  PROC DrawPart12()
    MoveL Offs(pOrigin,114.48,92.02,0.00),v60,z0,tPen\WObj:=wPaper;
    MoveL Offs(pOrigin,115.12,91.91,0.00),v40,z0,tPen\WObj:=wPaper;
    MoveL Offs(pOrigin,117.03,89.57,0.00),v40,z0,tPen\WObj:=wPaper;
    MoveL Offs(pOrigin,121.07,85.96,0.00),v40,z0,tPen\WObj:=wPaper;
    MoveL Offs(pOrigin,120.75,85.22,0.00),v40,z0,tPen\WObj:=wPaper;
    MoveL Offs(pOrigin,121.28,84.47,0.00),v40,fine,tPen\WObj:=wPaper;
    MoveL Offs(pOrigin,121.28,84.47,6.00),v60,z5,tPen\WObj:=wPaper;
    MoveL Offs(pOrigin,128.51,83.73,6.00),vTravel,z5,tPen\WObj:=wPaper;
    MoveL Offs(pOrigin,128.51,83.73,0.00),v60,z0,tPen\WObj:=wPaper;
    MoveL Offs(pOrigin,131.80,86.49,0.00),v40,z0,tPen\WObj:=wPaper;
    MoveL Offs(pOrigin,134.03,89.36,0.00),v40,fine,tPen\WObj:=wPaper;
    MoveL Offs(pOrigin,134.03,89.36,6.00),v60,z5,tPen\WObj:=wPaper;
    MoveL Offs(pOrigin,132.23,86.92,6.00),vTravel,z5,tPen\WObj:=wPaper;
    MoveL Offs(pOrigin,132.23,86.92,0.00),v60,z0,tPen\WObj:=wPaper;
    MoveL Offs(pOrigin,132.54,87.24,0.00),v40,z0,tPen\WObj:=wPaper;
    MoveL Offs(pOrigin,132.23,86.92,0.00),v40,fine,tPen\WObj:=wPaper;
    MoveL Offs(pOrigin,132.23,86.92,6.00),v60,z5,tPen\WObj:=wPaper;
    MoveL Offs(pOrigin,137.11,89.89,6.00),vTravel,z5,tPen\WObj:=wPaper;
    MoveL Offs(pOrigin,137.11,89.89,0.00),v60,z0,tPen\WObj:=wPaper;
    MoveL Offs(pOrigin,137.75,90.74,0.00),v40,fine,tPen\WObj:=wPaper;
    MoveL Offs(pOrigin,137.75,90.74,6.00),v60,z5,tPen\WObj:=wPaper;
    MoveL Offs(pOrigin,134.77,96.91,6.00),vTravel,z5,tPen\WObj:=wPaper;
    MoveL Offs(pOrigin,134.77,96.91,0.00),v60,z0,tPen\WObj:=wPaper;
    MoveL Offs(pOrigin,130.74,95.21,0.00),v40,fine,tPen\WObj:=wPaper;
    MoveL Offs(pOrigin,130.74,95.21,6.00),v60,z5,tPen\WObj:=wPaper;
    MoveL Offs(pOrigin,131.06,119.64,6.00),vTravel,z5,tPen\WObj:=wPaper;
    MoveL Offs(pOrigin,131.06,119.64,0.00),v60,z0,tPen\WObj:=wPaper;
    MoveL Offs(pOrigin,131.48,121.34,0.00),v40,z0,tPen\WObj:=wPaper;
    MoveL Offs(pOrigin,131.27,121.03,0.00),v40,z0,tPen\WObj:=wPaper;
    MoveL Offs(pOrigin,131.69,121.34,0.00),v40,z0,tPen\WObj:=wPaper;
    MoveL Offs(pOrigin,132.65,121.34,0.00),v40,z0,tPen\WObj:=wPaper;
    MoveL Offs(pOrigin,132.65,121.34,0.00),v40,z0,tPen\WObj:=wPaper;
    MoveL Offs(pOrigin,133.07,122.62,0.00),v40,z0,tPen\WObj:=wPaper;
    MoveL Offs(pOrigin,132.44,122.94,0.00),v40,fine,tPen\WObj:=wPaper;
    MoveL Offs(pOrigin,132.44,122.94,6.00),v60,z5,tPen\WObj:=wPaper;
    MoveL Offs(pOrigin,130.74,123.04,6.00),vTravel,z5,tPen\WObj:=wPaper;
    MoveL Offs(pOrigin,130.74,123.04,0.00),v60,z0,tPen\WObj:=wPaper;
    MoveL Offs(pOrigin,130.84,121.77,0.00),v40,z0,tPen\WObj:=wPaper;
    MoveL Offs(pOrigin,130.42,121.56,0.00),v40,z0,tPen\WObj:=wPaper;
    MoveL Offs(pOrigin,130.42,121.56,0.00),v40,z0,tPen\WObj:=wPaper;
    MoveL Offs(pOrigin,129.04,121.66,0.00),v40,fine,tPen\WObj:=wPaper;
    MoveL Offs(pOrigin,129.04,121.66,6.00),v60,z5,tPen\WObj:=wPaper;
    MoveL Offs(pOrigin,127.66,121.66,6.00),vTravel,z5,tPen\WObj:=wPaper;
    MoveL Offs(pOrigin,127.66,121.66,0.00),v60,z0,tPen\WObj:=wPaper;
    MoveL Offs(pOrigin,127.62,120.28,0.00),v40,z0,tPen\WObj:=wPaper;
    MoveL Offs(pOrigin,126.91,120.39,0.00),v40,z0,tPen\WObj:=wPaper;
    MoveL Offs(pOrigin,126.91,120.39,0.00),v40,z0,tPen\WObj:=wPaper;
    MoveL Offs(pOrigin,126.91,121.77,0.00),v40,z0,tPen\WObj:=wPaper;
    MoveL Offs(pOrigin,126.91,121.77,0.00),v40,z0,tPen\WObj:=wPaper;
    MoveL Offs(pOrigin,125.64,121.66,0.00),v40,z0,tPen\WObj:=wPaper;
    MoveL Offs(pOrigin,125.64,121.66,0.00),v40,z0,tPen\WObj:=wPaper;
    MoveL Offs(pOrigin,125.60,121.03,0.00),v40,z0,tPen\WObj:=wPaper;
    MoveL Offs(pOrigin,124.68,120.00,0.00),v40,z0,tPen\WObj:=wPaper;
    MoveL Offs(pOrigin,124.29,120.07,0.00),v40,z0,tPen\WObj:=wPaper;
    MoveL Offs(pOrigin,124.04,121.13,0.00),v40,z0,tPen\WObj:=wPaper;
    MoveL Offs(pOrigin,124.26,121.24,0.00),v40,z0,tPen\WObj:=wPaper;
    MoveL Offs(pOrigin,125.64,121.66,0.00),v40,z0,tPen\WObj:=wPaper;
    MoveL Offs(pOrigin,125.64,120.92,0.00),v40,z0,tPen\WObj:=wPaper;
    MoveL Offs(pOrigin,126.28,120.32,0.00),v40,z0,tPen\WObj:=wPaper;
    MoveL Offs(pOrigin,126.91,120.39,0.00),v40,fine,tPen\WObj:=wPaper;
    MoveL Offs(pOrigin,126.91,120.39,6.00),v60,z5,tPen\WObj:=wPaper;
    MoveL Offs(pOrigin,125.64,120.92,6.00),vTravel,z5,tPen\WObj:=wPaper;
    MoveL Offs(pOrigin,125.64,120.92,0.00),v60,z0,tPen\WObj:=wPaper;
    MoveL Offs(pOrigin,124.89,120.18,0.00),v40,fine,tPen\WObj:=wPaper;
    MoveL Offs(pOrigin,124.89,120.18,6.00),v60,z5,tPen\WObj:=wPaper;
    MoveL Offs(pOrigin,124.47,121.56,6.00),vTravel,z5,tPen\WObj:=wPaper;
    MoveL Offs(pOrigin,124.47,121.56,0.00),v60,z0,tPen\WObj:=wPaper;
    MoveL Offs(pOrigin,123.51,122.62,0.00),v40,z0,tPen\WObj:=wPaper;
    MoveL Offs(pOrigin,123.41,122.62,0.00),v40,z0,tPen\WObj:=wPaper;
    MoveL Offs(pOrigin,121.49,122.19,0.00),v40,z0,tPen\WObj:=wPaper;
    MoveL Offs(pOrigin,120.22,121.17,0.00),v40,z0,tPen\WObj:=wPaper;
    MoveL Offs(pOrigin,119.69,121.13,0.00),v40,z0,tPen\WObj:=wPaper;
    MoveL Offs(pOrigin,119.69,121.13,0.00),v40,z0,tPen\WObj:=wPaper;
    MoveL Offs(pOrigin,120.11,121.88,0.00),v40,z0,tPen\WObj:=wPaper;
    MoveL Offs(pOrigin,119.90,122.90,0.00),v40,z0,tPen\WObj:=wPaper;
    MoveL Offs(pOrigin,118.41,123.47,0.00),v40,z0,tPen\WObj:=wPaper;
    MoveL Offs(pOrigin,117.35,123.15,0.00),v40,z0,tPen\WObj:=wPaper;
    MoveL Offs(pOrigin,116.22,123.93,0.00),v40,z0,tPen\WObj:=wPaper;
    MoveL Offs(pOrigin,115.97,125.17,0.00),v40,z0,tPen\WObj:=wPaper;
    MoveL Offs(pOrigin,116.61,126.76,0.00),v40,fine,tPen\WObj:=wPaper;
    MoveL Offs(pOrigin,116.61,126.76,6.00),v60,z5,tPen\WObj:=wPaper;
    MoveL Offs(pOrigin,115.65,125.70,6.00),vTravel,z5,tPen\WObj:=wPaper;
    MoveL Offs(pOrigin,115.65,125.70,0.00),v60,z0,tPen\WObj:=wPaper;
    MoveL Offs(pOrigin,111.61,119.54,0.00),v40,fine,tPen\WObj:=wPaper;
    MoveL Offs(pOrigin,111.61,119.54,6.00),v60,z5,tPen\WObj:=wPaper;
    MoveL Offs(pOrigin,114.27,118.79,6.00),vTravel,z5,tPen\WObj:=wPaper;
    MoveL Offs(pOrigin,114.27,118.79,0.00),v60,z0,tPen\WObj:=wPaper;
    MoveL Offs(pOrigin,114.69,119.25,0.00),v40,z0,tPen\WObj:=wPaper;
    MoveL Offs(pOrigin,115.97,119.57,0.00),v40,z0,tPen\WObj:=wPaper;
    MoveL Offs(pOrigin,116.71,120.28,0.00),v40,z0,tPen\WObj:=wPaper;
    MoveL Offs(pOrigin,116.71,120.28,0.00),v40,z0,tPen\WObj:=wPaper;
    MoveL Offs(pOrigin,117.35,120.28,0.00),v40,z0,tPen\WObj:=wPaper;
    MoveL Offs(pOrigin,117.67,120.71,0.00),v40,z0,tPen\WObj:=wPaper;
    MoveL Offs(pOrigin,117.67,120.71,0.00),v40,z0,tPen\WObj:=wPaper;
    MoveL Offs(pOrigin,118.94,120.81,0.00),v40,z0,tPen\WObj:=wPaper;
    MoveL Offs(pOrigin,119.58,120.32,0.00),v40,z0,tPen\WObj:=wPaper;
    MoveL Offs(pOrigin,119.51,119.54,0.00),v40,z0,tPen\WObj:=wPaper;
    MoveL Offs(pOrigin,119.90,119.50,0.00),v40,z0,tPen\WObj:=wPaper;
    MoveL Offs(pOrigin,119.97,119.96,0.00),v40,z0,tPen\WObj:=wPaper;
    MoveL Offs(pOrigin,119.58,120.32,0.00),v40,z0,tPen\WObj:=wPaper;
    MoveL Offs(pOrigin,120.01,119.54,0.00),v40,z0,tPen\WObj:=wPaper;
    MoveL Offs(pOrigin,120.79,119.75,0.00),v40,z0,tPen\WObj:=wPaper;
    MoveL Offs(pOrigin,120.75,120.81,0.00),v40,fine,tPen\WObj:=wPaper;
    MoveL Offs(pOrigin,120.75,120.81,6.00),v60,z5,tPen\WObj:=wPaper;
    MoveL Offs(pOrigin,118.31,119.11,6.00),vTravel,z5,tPen\WObj:=wPaper;
    MoveL Offs(pOrigin,118.31,119.11,0.00),v60,z0,tPen\WObj:=wPaper;
    MoveL Offs(pOrigin,117.46,120.28,0.00),v40,fine,tPen\WObj:=wPaper;
    MoveL Offs(pOrigin,117.46,120.28,6.00),v60,z5,tPen\WObj:=wPaper;
    MoveL Offs(pOrigin,117.03,118.26,6.00),vTravel,z5,tPen\WObj:=wPaper;
    MoveL Offs(pOrigin,117.03,118.26,0.00),v60,z0,tPen\WObj:=wPaper;
    MoveL Offs(pOrigin,116.29,117.73,0.00),v40,z0,tPen\WObj:=wPaper;
    MoveL Offs(pOrigin,115.44,117.73,0.00),v40,z0,tPen\WObj:=wPaper;
    MoveL Offs(pOrigin,114.27,118.79,0.00),v40,z0,tPen\WObj:=wPaper;
    MoveL Offs(pOrigin,114.27,118.79,0.00),v40,z0,tPen\WObj:=wPaper;
    MoveL Offs(pOrigin,113.21,117.94,0.00),v40,z0,tPen\WObj:=wPaper;
    MoveL Offs(pOrigin,113.74,116.03,0.00),v40,fine,tPen\WObj:=wPaper;
    MoveL Offs(pOrigin,113.74,116.03,6.00),v60,z5,tPen\WObj:=wPaper;
    MoveL Offs(pOrigin,116.61,117.84,6.00),vTravel,z5,tPen\WObj:=wPaper;
    MoveL Offs(pOrigin,116.61,117.84,0.00),v60,z0,tPen\WObj:=wPaper;
    MoveL Offs(pOrigin,130.21,119.32,0.00),v40,z0,tPen\WObj:=wPaper;
  ENDPROC

  PROC DrawPart13()
    MoveL Offs(pOrigin,131.80,119.68,0.00),v40,z0,tPen\WObj:=wPaper;
    MoveL Offs(pOrigin,132.76,120.71,0.00),v40,z0,tPen\WObj:=wPaper;
    MoveL Offs(pOrigin,132.76,120.71,0.00),v40,z0,tPen\WObj:=wPaper;
    MoveL Offs(pOrigin,131.80,119.75,0.00),v40,fine,tPen\WObj:=wPaper;
    MoveL Offs(pOrigin,131.80,119.75,6.00),v60,z5,tPen\WObj:=wPaper;
    MoveL Offs(pOrigin,134.56,122.41,6.00),vTravel,z5,tPen\WObj:=wPaper;
    MoveL Offs(pOrigin,134.56,122.41,0.00),v60,z0,tPen\WObj:=wPaper;
    MoveL Offs(pOrigin,128.61,127.40,0.00),v40,z0,tPen\WObj:=wPaper;
    MoveL Offs(pOrigin,127.55,127.72,0.00),v40,z0,tPen\WObj:=wPaper;
    MoveL Offs(pOrigin,128.19,126.12,0.00),v40,z0,tPen\WObj:=wPaper;
    MoveL Offs(pOrigin,127.90,125.06,0.00),v40,z0,tPen\WObj:=wPaper;
    MoveL Offs(pOrigin,127.23,124.39,0.00),v40,z0,tPen\WObj:=wPaper;
    MoveL Offs(pOrigin,126.38,124.32,0.00),v40,z0,tPen\WObj:=wPaper;
    MoveL Offs(pOrigin,126.38,124.32,0.00),v40,z0,tPen\WObj:=wPaper;
    MoveL Offs(pOrigin,126.06,124.64,0.00),v40,z0,tPen\WObj:=wPaper;
    MoveL Offs(pOrigin,125.00,124.25,0.00),v40,z0,tPen\WObj:=wPaper;
    MoveL Offs(pOrigin,123.51,122.72,0.00),v40,z0,tPen\WObj:=wPaper;
    MoveL Offs(pOrigin,123.94,123.47,0.00),v40,z0,tPen\WObj:=wPaper;
    MoveL Offs(pOrigin,124.26,123.79,0.00),v40,z0,tPen\WObj:=wPaper;
    MoveL Offs(pOrigin,123.94,123.47,0.00),v40,fine,tPen\WObj:=wPaper;
    MoveL Offs(pOrigin,123.94,123.47,6.00),v60,z5,tPen\WObj:=wPaper;
    MoveL Offs(pOrigin,127.66,121.66,6.00),vTravel,z5,tPen\WObj:=wPaper;
    MoveL Offs(pOrigin,127.66,121.66,0.00),v60,z0,tPen\WObj:=wPaper;
    MoveL Offs(pOrigin,129.00,121.77,0.00),v40,z0,tPen\WObj:=wPaper;
    MoveL Offs(pOrigin,129.00,122.51,0.00),v40,z0,tPen\WObj:=wPaper;
    MoveL Offs(pOrigin,128.51,123.26,0.00),v40,fine,tPen\WObj:=wPaper;
    MoveL Offs(pOrigin,128.51,123.26,6.00),v60,z5,tPen\WObj:=wPaper;
    MoveL Offs(pOrigin,129.99,131.76,6.00),vTravel,z5,tPen\WObj:=wPaper;
    MoveL Offs(pOrigin,129.99,131.76,0.00),v60,z0,tPen\WObj:=wPaper;
    MoveL Offs(pOrigin,127.66,132.36,0.00),v40,z0,tPen\WObj:=wPaper;
    MoveL Offs(pOrigin,125.96,133.24,0.00),v40,z0,tPen\WObj:=wPaper;
    MoveL Offs(pOrigin,127.02,133.56,0.00),v40,z0,tPen\WObj:=wPaper;
    MoveL Offs(pOrigin,128.82,133.14,0.00),v40,fine,tPen\WObj:=wPaper;
    MoveL Offs(pOrigin,128.82,133.14,6.00),v60,z5,tPen\WObj:=wPaper;
    MoveL Offs(pOrigin,129.46,135.37,6.00),vTravel,z5,tPen\WObj:=wPaper;
    MoveL Offs(pOrigin,129.46,135.37,0.00),v60,z0,tPen\WObj:=wPaper;
    MoveL Offs(pOrigin,128.75,135.51,0.00),v40,z0,tPen\WObj:=wPaper;
    MoveL Offs(pOrigin,128.72,136.25,0.00),v40,z0,tPen\WObj:=wPaper;
    MoveL Offs(pOrigin,129.78,135.48,0.00),v40,z0,tPen\WObj:=wPaper;
    MoveL Offs(pOrigin,130.52,136.22,0.00),v40,z0,tPen\WObj:=wPaper;
    MoveL Offs(pOrigin,130.10,136.71,0.00),v40,z0,tPen\WObj:=wPaper;
    MoveL Offs(pOrigin,129.14,136.75,0.00),v40,z0,tPen\WObj:=wPaper;
    MoveL Offs(pOrigin,127.87,136.25,0.00),v40,z0,tPen\WObj:=wPaper;
    MoveL Offs(pOrigin,126.81,135.26,0.00),v40,z0,tPen\WObj:=wPaper;
    MoveL Offs(pOrigin,126.81,135.26,0.00),v40,z0,tPen\WObj:=wPaper;
    MoveL Offs(pOrigin,126.91,134.84,0.00),v40,z0,tPen\WObj:=wPaper;
    MoveL Offs(pOrigin,126.38,134.62,0.00),v40,z0,tPen\WObj:=wPaper;
    MoveL Offs(pOrigin,126.91,134.73,0.00),v40,z0,tPen\WObj:=wPaper;
    MoveL Offs(pOrigin,129.04,134.73,0.00),v40,z0,tPen\WObj:=wPaper;
    MoveL Offs(pOrigin,129.57,135.33,0.00),v40,z0,tPen\WObj:=wPaper;
    MoveL Offs(pOrigin,130.38,135.62,0.00),v40,z0,tPen\WObj:=wPaper;
    MoveL Offs(pOrigin,130.52,136.22,0.00),v40,z0,tPen\WObj:=wPaper;
    MoveL Offs(pOrigin,130.52,136.22,0.00),v40,z0,tPen\WObj:=wPaper;
    MoveL Offs(pOrigin,131.48,136.64,0.00),v40,z0,tPen\WObj:=wPaper;
    MoveL Offs(pOrigin,133.18,135.90,0.00),v40,z0,tPen\WObj:=wPaper;
    MoveL Offs(pOrigin,133.93,135.90,0.00),v40,z0,tPen\WObj:=wPaper;
    MoveL Offs(pOrigin,133.93,135.90,0.00),v40,z0,tPen\WObj:=wPaper;
    MoveL Offs(pOrigin,134.46,136.11,0.00),v40,z0,tPen\WObj:=wPaper;
    MoveL Offs(pOrigin,135.20,135.79,0.00),v40,fine,tPen\WObj:=wPaper;
    MoveL Offs(pOrigin,135.20,135.79,6.00),v60,z5,tPen\WObj:=wPaper;
    MoveL Offs(pOrigin,136.37,135.48,6.00),vTravel,z5,tPen\WObj:=wPaper;
    MoveL Offs(pOrigin,136.37,135.48,0.00),v60,z0,tPen\WObj:=wPaper;
    MoveL Offs(pOrigin,134.88,135.37,0.00),v40,z0,tPen\WObj:=wPaper;
    MoveL Offs(pOrigin,133.93,135.90,0.00),v40,z0,tPen\WObj:=wPaper;
    MoveL Offs(pOrigin,133.93,136.11,0.00),v40,z0,tPen\WObj:=wPaper;
    MoveL Offs(pOrigin,133.50,136.68,0.00),v40,z0,tPen\WObj:=wPaper;
    MoveL Offs(pOrigin,132.44,137.18,0.00),v40,z0,tPen\WObj:=wPaper;
    MoveL Offs(pOrigin,128.61,137.49,0.00),v40,z0,tPen\WObj:=wPaper;
    MoveL Offs(pOrigin,127.12,137.14,0.00),v40,z0,tPen\WObj:=wPaper;
    MoveL Offs(pOrigin,125.43,135.48,0.00),v40,z0,tPen\WObj:=wPaper;
    MoveL Offs(pOrigin,124.68,135.16,0.00),v40,z0,tPen\WObj:=wPaper;
    MoveL Offs(pOrigin,124.57,135.37,0.00),v40,z0,tPen\WObj:=wPaper;
    MoveL Offs(pOrigin,125.53,135.79,0.00),v40,fine,tPen\WObj:=wPaper;
    MoveL Offs(pOrigin,125.53,135.79,6.00),v60,z5,tPen\WObj:=wPaper;
    MoveL Offs(pOrigin,123.62,134.41,6.00),vTravel,z5,tPen\WObj:=wPaper;
    MoveL Offs(pOrigin,123.62,134.41,0.00),v60,z0,tPen\WObj:=wPaper;
    MoveL Offs(pOrigin,123.30,135.37,0.00),v40,z0,tPen\WObj:=wPaper;
    MoveL Offs(pOrigin,123.37,136.64,0.00),v40,z0,tPen\WObj:=wPaper;
    MoveL Offs(pOrigin,124.79,137.85,0.00),v40,z0,tPen\WObj:=wPaper;
    MoveL Offs(pOrigin,131.80,139.19,0.00),v40,z0,tPen\WObj:=wPaper;
    MoveL Offs(pOrigin,134.14,139.09,0.00),v40,z0,tPen\WObj:=wPaper;
    MoveL Offs(pOrigin,135.41,138.34,0.00),v40,fine,tPen\WObj:=wPaper;
    MoveL Offs(pOrigin,135.41,138.34,6.00),v60,z5,tPen\WObj:=wPaper;
    MoveL Offs(pOrigin,137.54,138.88,6.00),vTravel,z5,tPen\WObj:=wPaper;
    MoveL Offs(pOrigin,137.54,138.88,0.00),v60,z0,tPen\WObj:=wPaper;
    MoveL Offs(pOrigin,138.18,137.18,0.00),v40,z0,tPen\WObj:=wPaper;
    MoveL Offs(pOrigin,138.18,137.18,0.00),v40,z0,tPen\WObj:=wPaper;
    MoveL Offs(pOrigin,138.18,133.67,0.00),v40,z0,tPen\WObj:=wPaper;
    MoveL Offs(pOrigin,137.43,131.54,0.00),v40,z0,tPen\WObj:=wPaper;
    MoveL Offs(pOrigin,135.52,130.55,0.00),v40,z0,tPen\WObj:=wPaper;
    MoveL Offs(pOrigin,133.18,129.95,0.00),v40,z0,tPen\WObj:=wPaper;
    MoveL Offs(pOrigin,130.10,129.52,0.00),v40,z0,tPen\WObj:=wPaper;
    MoveL Offs(pOrigin,127.44,129.52,0.00),v40,z0,tPen\WObj:=wPaper;
    MoveL Offs(pOrigin,125.96,129.91,0.00),v40,z0,tPen\WObj:=wPaper;
    MoveL Offs(pOrigin,124.04,131.86,0.00),v40,z0,tPen\WObj:=wPaper;
    MoveL Offs(pOrigin,123.26,133.03,0.00),v40,z0,tPen\WObj:=wPaper;
    MoveL Offs(pOrigin,122.63,135.37,0.00),v40,z0,tPen\WObj:=wPaper;
    MoveL Offs(pOrigin,120.96,135.69,0.00),v40,z0,tPen\WObj:=wPaper;
    MoveL Offs(pOrigin,119.05,135.19,0.00),v40,z0,tPen\WObj:=wPaper;
    MoveL Offs(pOrigin,118.62,134.73,0.00),v40,z0,tPen\WObj:=wPaper;
    MoveL Offs(pOrigin,118.84,133.77,0.00),v40,z0,tPen\WObj:=wPaper;
    MoveL Offs(pOrigin,118.84,133.56,0.00),v40,z0,tPen\WObj:=wPaper;
    MoveL Offs(pOrigin,118.73,132.61,0.00),v40,z0,tPen\WObj:=wPaper;
    MoveL Offs(pOrigin,118.73,132.61,0.00),v40,z0,tPen\WObj:=wPaper;
    MoveL Offs(pOrigin,118.31,131.23,0.00),v40,z0,tPen\WObj:=wPaper;
    MoveL Offs(pOrigin,118.31,131.01,0.00),v40,z0,tPen\WObj:=wPaper;
    MoveL Offs(pOrigin,117.46,129.31,0.00),v40,z0,tPen\WObj:=wPaper;
    MoveL Offs(pOrigin,116.07,128.32,0.00),v40,z0,tPen\WObj:=wPaper;
    MoveL Offs(pOrigin,112.78,127.51,0.00),v40,z0,tPen\WObj:=wPaper;
    MoveL Offs(pOrigin,108.53,127.19,0.00),v40,z0,tPen\WObj:=wPaper;
    MoveL Offs(pOrigin,106.72,127.40,0.00),v40,z0,tPen\WObj:=wPaper;
    MoveL Offs(pOrigin,105.45,128.04,0.00),v40,z0,tPen\WObj:=wPaper;
    MoveL Offs(pOrigin,104.46,129.63,0.00),v40,z0,tPen\WObj:=wPaper;
    MoveL Offs(pOrigin,103.54,132.18,0.00),v40,z0,tPen\WObj:=wPaper;
    MoveL Offs(pOrigin,103.54,132.18,0.00),v40,z0,tPen\WObj:=wPaper;
    MoveL Offs(pOrigin,104.07,135.16,0.00),v40,z0,tPen\WObj:=wPaper;
    MoveL Offs(pOrigin,104.07,135.16,0.00),v40,z0,tPen\WObj:=wPaper;
    MoveL Offs(pOrigin,105.34,135.94,0.00),v40,z0,tPen\WObj:=wPaper;
    MoveL Offs(pOrigin,109.17,137.28,0.00),v40,z0,tPen\WObj:=wPaper;
    MoveL Offs(pOrigin,113.74,137.71,0.00),v40,z0,tPen\WObj:=wPaper;
  ENDPROC

  PROC DrawPart14()
    MoveL Offs(pOrigin,115.01,138.24,0.00),v40,z0,tPen\WObj:=wPaper;
    MoveL Offs(pOrigin,114.80,137.49,0.00),v40,z0,tPen\WObj:=wPaper;
    MoveL Offs(pOrigin,117.78,136.75,0.00),v40,z0,tPen\WObj:=wPaper;
    MoveL Offs(pOrigin,117.99,137.07,0.00),v40,z0,tPen\WObj:=wPaper;
    MoveL Offs(pOrigin,117.78,136.64,0.00),v40,z0,tPen\WObj:=wPaper;
    MoveL Offs(pOrigin,118.09,136.32,0.00),v40,z0,tPen\WObj:=wPaper;
    MoveL Offs(pOrigin,118.09,136.32,0.00),v40,z0,tPen\WObj:=wPaper;
    MoveL Offs(pOrigin,118.31,136.75,0.00),v40,z0,tPen\WObj:=wPaper;
    MoveL Offs(pOrigin,117.99,137.28,0.00),v40,z0,tPen\WObj:=wPaper;
    MoveL Offs(pOrigin,118.09,139.62,0.00),v40,fine,tPen\WObj:=wPaper;
    MoveL Offs(pOrigin,118.09,139.62,6.00),v60,z5,tPen\WObj:=wPaper;
    MoveL Offs(pOrigin,118.09,136.32,6.00),vTravel,z5,tPen\WObj:=wPaper;
    MoveL Offs(pOrigin,118.09,136.32,0.00),v60,z0,tPen\WObj:=wPaper;
    MoveL Offs(pOrigin,118.41,135.79,0.00),v40,z0,tPen\WObj:=wPaper;
    MoveL Offs(pOrigin,120.75,136.43,0.00),v40,z0,tPen\WObj:=wPaper;
    MoveL Offs(pOrigin,122.45,136.32,0.00),v40,z0,tPen\WObj:=wPaper;
    MoveL Offs(pOrigin,122.88,137.35,0.00),v40,z0,tPen\WObj:=wPaper;
    MoveL Offs(pOrigin,125.21,139.02,0.00),v40,z0,tPen\WObj:=wPaper;
    MoveL Offs(pOrigin,127.02,139.62,0.00),v40,z0,tPen\WObj:=wPaper;
    MoveL Offs(pOrigin,132.12,140.26,0.00),v40,z0,tPen\WObj:=wPaper;
    MoveL Offs(pOrigin,135.94,139.73,0.00),v40,z0,tPen\WObj:=wPaper;
    MoveL Offs(pOrigin,137.54,138.88,0.00),v40,z0,tPen\WObj:=wPaper;
    MoveL Offs(pOrigin,137.54,138.88,0.00),v40,z0,tPen\WObj:=wPaper;
    MoveL Offs(pOrigin,139.66,139.09,0.00),v40,z0,tPen\WObj:=wPaper;
    MoveL Offs(pOrigin,139.66,139.09,0.00),v40,z0,tPen\WObj:=wPaper;
    MoveL Offs(pOrigin,139.63,138.45,0.00),v40,z0,tPen\WObj:=wPaper;
    MoveL Offs(pOrigin,138.71,138.02,0.00),v40,z0,tPen\WObj:=wPaper;
    MoveL Offs(pOrigin,138.18,137.18,0.00),v40,z0,tPen\WObj:=wPaper;
    MoveL Offs(pOrigin,139.77,137.92,0.00),v40,z0,tPen\WObj:=wPaper;
    MoveL Offs(pOrigin,139.66,138.34,0.00),v40,z0,tPen\WObj:=wPaper;
    MoveL Offs(pOrigin,139.98,137.92,0.00),v40,z0,tPen\WObj:=wPaper;
    MoveL Offs(pOrigin,142.43,137.81,0.00),v40,z0,tPen\WObj:=wPaper;
    MoveL Offs(pOrigin,142.21,138.56,0.00),v40,z0,tPen\WObj:=wPaper;
    MoveL Offs(pOrigin,140.41,138.45,0.00),v40,z0,tPen\WObj:=wPaper;
    MoveL Offs(pOrigin,139.66,139.09,0.00),v40,z0,tPen\WObj:=wPaper;
    MoveL Offs(pOrigin,141.15,139.09,0.00),v40,z0,tPen\WObj:=wPaper;
    MoveL Offs(pOrigin,141.57,139.51,0.00),v40,fine,tPen\WObj:=wPaper;
    MoveL Offs(pOrigin,141.57,139.51,6.00),v60,z5,tPen\WObj:=wPaper;
    MoveL Offs(pOrigin,142.74,140.79,6.00),vTravel,z5,tPen\WObj:=wPaper;
    MoveL Offs(pOrigin,142.74,140.79,0.00),v60,z0,tPen\WObj:=wPaper;
    MoveL Offs(pOrigin,140.94,143.23,0.00),v40,z0,tPen\WObj:=wPaper;
    MoveL Offs(pOrigin,140.94,143.23,0.00),v40,z0,tPen\WObj:=wPaper;
    MoveL Offs(pOrigin,139.66,145.78,0.00),v40,z0,tPen\WObj:=wPaper;
    MoveL Offs(pOrigin,139.45,144.93,0.00),v40,z0,tPen\WObj:=wPaper;
    MoveL Offs(pOrigin,140.41,143.44,0.00),v40,z0,tPen\WObj:=wPaper;
    MoveL Offs(pOrigin,140.94,143.23,0.00),v40,z0,tPen\WObj:=wPaper;
    MoveL Offs(pOrigin,140.73,142.38,0.00),v40,z0,tPen\WObj:=wPaper;
    MoveL Offs(pOrigin,141.15,141.32,0.00),v40,z0,tPen\WObj:=wPaper;
    MoveL Offs(pOrigin,141.15,141.32,0.00),v40,z0,tPen\WObj:=wPaper;
    MoveL Offs(pOrigin,142.43,141.21,0.00),v40,z0,tPen\WObj:=wPaper;
    MoveL Offs(pOrigin,142.74,140.79,0.00),v40,z0,tPen\WObj:=wPaper;
    MoveL Offs(pOrigin,144.44,140.15,0.00),v40,z0,tPen\WObj:=wPaper;
    MoveL Offs(pOrigin,144.44,140.15,0.00),v40,z0,tPen\WObj:=wPaper;
    MoveL Offs(pOrigin,145.40,140.57,0.00),v40,z0,tPen\WObj:=wPaper;
    MoveL Offs(pOrigin,146.36,140.47,0.00),v40,z0,tPen\WObj:=wPaper;
    MoveL Offs(pOrigin,145.82,139.90,0.00),v40,z0,tPen\WObj:=wPaper;
    MoveL Offs(pOrigin,145.08,139.73,0.00),v40,z0,tPen\WObj:=wPaper;
    MoveL Offs(pOrigin,144.44,140.15,0.00),v40,z0,tPen\WObj:=wPaper;
    MoveL Offs(pOrigin,144.66,141.21,0.00),v40,z0,tPen\WObj:=wPaper;
    MoveL Offs(pOrigin,143.27,141.85,0.00),v40,z0,tPen\WObj:=wPaper;
    MoveL Offs(pOrigin,143.17,142.81,0.00),v40,z0,tPen\WObj:=wPaper;
    MoveL Offs(pOrigin,143.17,142.81,0.00),v40,z0,tPen\WObj:=wPaper;
    MoveL Offs(pOrigin,141.68,144.19,0.00),v40,z0,tPen\WObj:=wPaper;
    MoveL Offs(pOrigin,141.47,145.04,0.00),v40,z0,tPen\WObj:=wPaper;
    MoveL Offs(pOrigin,141.47,145.04,0.00),v40,z0,tPen\WObj:=wPaper;
    MoveL Offs(pOrigin,140.65,146.52,0.00),v40,z0,tPen\WObj:=wPaper;
    MoveL Offs(pOrigin,141.26,147.06,0.00),v40,z0,tPen\WObj:=wPaper;
    MoveL Offs(pOrigin,141.26,147.06,0.00),v40,z0,tPen\WObj:=wPaper;
    MoveL Offs(pOrigin,143.27,145.53,0.00),v40,z0,tPen\WObj:=wPaper;
    MoveL Offs(pOrigin,143.59,145.68,0.00),v40,z0,tPen\WObj:=wPaper;
    MoveL Offs(pOrigin,143.49,145.46,0.00),v40,z0,tPen\WObj:=wPaper;
    MoveL Offs(pOrigin,145.93,145.68,0.00),v40,z0,tPen\WObj:=wPaper;
    MoveL Offs(pOrigin,146.46,146.31,0.00),v40,z0,tPen\WObj:=wPaper;
    MoveL Offs(pOrigin,146.46,146.31,0.00),v40,z0,tPen\WObj:=wPaper;
    MoveL Offs(pOrigin,144.23,146.70,0.00),v40,z0,tPen\WObj:=wPaper;
    MoveL Offs(pOrigin,143.31,147.48,0.00),v40,z0,tPen\WObj:=wPaper;
    MoveL Offs(pOrigin,143.70,147.69,0.00),v40,z0,tPen\WObj:=wPaper;
    MoveL Offs(pOrigin,144.76,147.48,0.00),v40,z0,tPen\WObj:=wPaper;
    MoveL Offs(pOrigin,147.10,148.23,0.00),v40,z0,tPen\WObj:=wPaper;
    MoveL Offs(pOrigin,147.10,148.23,0.00),v40,z0,tPen\WObj:=wPaper;
    MoveL Offs(pOrigin,147.21,149.18,0.00),v40,z0,tPen\WObj:=wPaper;
    MoveL Offs(pOrigin,147.21,149.18,0.00),v40,z0,tPen\WObj:=wPaper;
    MoveL Offs(pOrigin,148.16,149.50,0.00),v40,z0,tPen\WObj:=wPaper;
    MoveL Offs(pOrigin,148.16,149.50,0.00),v40,z0,tPen\WObj:=wPaper;
    MoveL Offs(pOrigin,148.45,148.44,0.00),v40,z0,tPen\WObj:=wPaper;
    MoveL Offs(pOrigin,147.10,148.23,0.00),v40,z0,tPen\WObj:=wPaper;
    MoveL Offs(pOrigin,147.21,149.18,0.00),v40,z0,tPen\WObj:=wPaper;
    MoveL Offs(pOrigin,145.08,149.07,0.00),v40,z0,tPen\WObj:=wPaper;
    MoveL Offs(pOrigin,143.81,149.61,0.00),v40,z0,tPen\WObj:=wPaper;
    MoveL Offs(pOrigin,143.81,149.61,0.00),v40,z0,tPen\WObj:=wPaper;
    MoveL Offs(pOrigin,143.91,150.21,0.00),v40,z0,tPen\WObj:=wPaper;
    MoveL Offs(pOrigin,145.51,150.03,0.00),v40,z0,tPen\WObj:=wPaper;
    MoveL Offs(pOrigin,146.25,150.46,0.00),v40,z0,tPen\WObj:=wPaper;
    MoveL Offs(pOrigin,146.25,150.46,0.00),v40,z0,tPen\WObj:=wPaper;
    MoveL Offs(pOrigin,148.27,151.20,0.00),v40,z0,tPen\WObj:=wPaper;
    MoveL Offs(pOrigin,148.27,151.20,0.00),v40,z0,tPen\WObj:=wPaper;
    MoveL Offs(pOrigin,148.06,152.37,0.00),v40,z0,tPen\WObj:=wPaper;
    MoveL Offs(pOrigin,148.06,152.37,0.00),v40,z0,tPen\WObj:=wPaper;
    MoveL Offs(pOrigin,146.89,152.05,0.00),v40,z0,tPen\WObj:=wPaper;
    MoveL Offs(pOrigin,146.68,152.37,0.00),v40,z0,tPen\WObj:=wPaper;
    MoveL Offs(pOrigin,147.21,152.83,0.00),v40,z0,tPen\WObj:=wPaper;
    MoveL Offs(pOrigin,148.06,152.90,0.00),v40,z0,tPen\WObj:=wPaper;
    MoveL Offs(pOrigin,148.06,152.90,0.00),v40,z0,tPen\WObj:=wPaper;
    MoveL Offs(pOrigin,147.84,154.07,0.00),v40,z0,tPen\WObj:=wPaper;
    MoveL Offs(pOrigin,147.84,154.07,0.00),v40,z0,tPen\WObj:=wPaper;
    MoveL Offs(pOrigin,147.56,155.34,0.00),v40,z0,tPen\WObj:=wPaper;
    MoveL Offs(pOrigin,146.78,155.77,0.00),v40,z0,tPen\WObj:=wPaper;
    MoveL Offs(pOrigin,146.53,156.73,0.00),v40,z0,tPen\WObj:=wPaper;
    MoveL Offs(pOrigin,146.07,157.15,0.00),v40,z0,tPen\WObj:=wPaper;
    MoveL Offs(pOrigin,145.93,159.06,0.00),v40,z0,tPen\WObj:=wPaper;
    MoveL Offs(pOrigin,145.40,158.96,0.00),v40,z0,tPen\WObj:=wPaper;
    MoveL Offs(pOrigin,145.44,158.11,0.00),v40,z0,tPen\WObj:=wPaper;
    MoveL Offs(pOrigin,145.93,157.79,0.00),v40,z0,tPen\WObj:=wPaper;
    MoveL Offs(pOrigin,146.04,157.04,0.00),v40,z0,tPen\WObj:=wPaper;
    MoveL Offs(pOrigin,145.51,155.77,0.00),v40,z0,tPen\WObj:=wPaper;
    MoveL Offs(pOrigin,145.51,155.77,0.00),v40,z0,tPen\WObj:=wPaper;
    MoveL Offs(pOrigin,144.94,156.19,0.00),v40,z0,tPen\WObj:=wPaper;
    MoveL Offs(pOrigin,143.56,158.74,0.00),v40,z0,tPen\WObj:=wPaper;
    MoveL Offs(pOrigin,141.89,159.59,0.00),v40,z0,tPen\WObj:=wPaper;
    MoveL Offs(pOrigin,140.09,159.35,0.00),v40,z0,tPen\WObj:=wPaper;
  ENDPROC

  PROC DrawPart15()
    MoveL Offs(pOrigin,137.75,158.00,0.00),v40,z0,tPen\WObj:=wPaper;
    MoveL Offs(pOrigin,135.73,158.00,0.00),v40,z0,tPen\WObj:=wPaper;
    MoveL Offs(pOrigin,135.31,158.32,0.00),v40,z0,tPen\WObj:=wPaper;
    MoveL Offs(pOrigin,135.31,158.32,0.00),v40,z0,tPen\WObj:=wPaper;
    MoveL Offs(pOrigin,132.97,158.21,0.00),v40,z0,tPen\WObj:=wPaper;
    MoveL Offs(pOrigin,130.42,157.36,0.00),v40,fine,tPen\WObj:=wPaper;
    MoveL Offs(pOrigin,130.42,157.36,6.00),v60,z5,tPen\WObj:=wPaper;
    MoveL Offs(pOrigin,129.04,157.68,6.00),vTravel,z5,tPen\WObj:=wPaper;
    MoveL Offs(pOrigin,129.04,157.68,0.00),v60,z0,tPen\WObj:=wPaper;
    MoveL Offs(pOrigin,130.84,158.85,0.00),v40,z0,tPen\WObj:=wPaper;
    MoveL Offs(pOrigin,134.03,159.27,0.00),v40,z0,tPen\WObj:=wPaper;
    MoveL Offs(pOrigin,134.67,160.12,0.00),v40,z0,tPen\WObj:=wPaper;
    MoveL Offs(pOrigin,135.62,160.76,0.00),v40,z0,tPen\WObj:=wPaper;
    MoveL Offs(pOrigin,135.62,160.76,0.00),v40,z0,tPen\WObj:=wPaper;
    MoveL Offs(pOrigin,137.86,161.61,0.00),v40,fine,tPen\WObj:=wPaper;
    MoveL Offs(pOrigin,137.86,161.61,6.00),v60,z5,tPen\WObj:=wPaper;
    MoveL Offs(pOrigin,136.69,162.78,6.00),vTravel,z5,tPen\WObj:=wPaper;
    MoveL Offs(pOrigin,136.69,162.78,0.00),v60,z0,tPen\WObj:=wPaper;
    MoveL Offs(pOrigin,134.46,161.19,0.00),v40,z0,tPen\WObj:=wPaper;
    MoveL Offs(pOrigin,134.46,161.19,0.00),v40,z0,tPen\WObj:=wPaper;
    MoveL Offs(pOrigin,135.52,161.22,0.00),v40,z0,tPen\WObj:=wPaper;
    MoveL Offs(pOrigin,139.56,163.42,0.00),v40,z0,tPen\WObj:=wPaper;
    MoveL Offs(pOrigin,141.86,163.52,0.00),v40,z0,tPen\WObj:=wPaper;
    MoveL Offs(pOrigin,141.75,164.02,0.00),v40,z0,tPen\WObj:=wPaper;
    MoveL Offs(pOrigin,140.30,164.69,0.00),v40,z0,tPen\WObj:=wPaper;
    MoveL Offs(pOrigin,139.66,164.38,0.00),v40,z0,tPen\WObj:=wPaper;
    MoveL Offs(pOrigin,140.09,164.69,0.00),v40,z0,tPen\WObj:=wPaper;
    MoveL Offs(pOrigin,139.45,165.01,0.00),v40,z0,tPen\WObj:=wPaper;
    MoveL Offs(pOrigin,137.86,164.91,0.00),v40,z0,tPen\WObj:=wPaper;
    MoveL Offs(pOrigin,136.37,164.30,0.00),v40,z0,tPen\WObj:=wPaper;
    MoveL Offs(pOrigin,133.71,162.32,0.00),v40,z0,tPen\WObj:=wPaper;
    MoveL Offs(pOrigin,131.69,162.04,0.00),v40,z0,tPen\WObj:=wPaper;
    MoveL Offs(pOrigin,131.69,162.04,0.00),v40,z0,tPen\WObj:=wPaper;
    MoveL Offs(pOrigin,132.65,163.31,0.00),v40,z0,tPen\WObj:=wPaper;
    MoveL Offs(pOrigin,132.65,163.31,0.00),v40,z0,tPen\WObj:=wPaper;
    MoveL Offs(pOrigin,134.77,165.65,0.00),v40,z0,tPen\WObj:=wPaper;
    MoveL Offs(pOrigin,134.03,165.12,0.00),v40,z0,tPen\WObj:=wPaper;
    MoveL Offs(pOrigin,133.71,166.39,0.00),v40,z0,tPen\WObj:=wPaper;
    MoveL Offs(pOrigin,133.71,166.82,0.00),v40,z0,tPen\WObj:=wPaper;
    MoveL Offs(pOrigin,132.65,169.26,0.00),v40,z0,tPen\WObj:=wPaper;
    MoveL Offs(pOrigin,132.65,169.26,0.00),v40,z0,tPen\WObj:=wPaper;
    MoveL Offs(pOrigin,133.61,169.05,0.00),v40,z0,tPen\WObj:=wPaper;
    MoveL Offs(pOrigin,133.61,169.05,0.00),v40,z0,tPen\WObj:=wPaper;
    MoveL Offs(pOrigin,134.14,168.09,0.00),v40,z0,tPen\WObj:=wPaper;
    MoveL Offs(pOrigin,134.14,168.09,0.00),v40,z0,tPen\WObj:=wPaper;
    MoveL Offs(pOrigin,133.71,166.82,0.00),v40,z0,tPen\WObj:=wPaper;
    MoveL Offs(pOrigin,133.71,166.82,0.00),v40,z0,tPen\WObj:=wPaper;
    MoveL Offs(pOrigin,131.91,163.52,0.00),v40,z0,tPen\WObj:=wPaper;
    MoveL Offs(pOrigin,131.91,163.52,0.00),v40,z0,tPen\WObj:=wPaper;
    MoveL Offs(pOrigin,130.74,162.85,0.00),v40,z0,tPen\WObj:=wPaper;
    MoveL Offs(pOrigin,129.78,162.78,0.00),v40,z0,tPen\WObj:=wPaper;
    MoveL Offs(pOrigin,129.78,162.78,0.00),v40,z0,tPen\WObj:=wPaper;
    MoveL Offs(pOrigin,131.45,165.12,0.00),v40,z0,tPen\WObj:=wPaper;
    MoveL Offs(pOrigin,131.80,167.67,0.00),v40,z0,tPen\WObj:=wPaper;
    MoveL Offs(pOrigin,131.06,169.26,0.00),v40,z0,tPen\WObj:=wPaper;
    MoveL Offs(pOrigin,129.57,170.96,0.00),v40,z0,tPen\WObj:=wPaper;
    MoveL Offs(pOrigin,129.57,170.96,0.00),v40,z0,tPen\WObj:=wPaper;
    MoveL Offs(pOrigin,131.48,170.54,0.00),v40,z0,tPen\WObj:=wPaper;
    MoveL Offs(pOrigin,131.48,170.54,0.00),v40,z0,tPen\WObj:=wPaper;
    MoveL Offs(pOrigin,132.65,169.26,0.00),v40,z0,tPen\WObj:=wPaper;
    MoveL Offs(pOrigin,132.97,170.22,0.00),v40,z0,tPen\WObj:=wPaper;
    MoveL Offs(pOrigin,133.71,169.69,0.00),v40,z0,tPen\WObj:=wPaper;
    MoveL Offs(pOrigin,133.71,169.69,0.00),v40,z0,tPen\WObj:=wPaper;
    MoveL Offs(pOrigin,136.05,168.27,0.00),v40,z0,tPen\WObj:=wPaper;
    MoveL Offs(pOrigin,137.54,166.43,0.00),v40,z0,tPen\WObj:=wPaper;
    MoveL Offs(pOrigin,140.41,165.79,0.00),v40,z0,tPen\WObj:=wPaper;
    MoveL Offs(pOrigin,142.21,164.80,0.00),v40,z0,tPen\WObj:=wPaper;
    MoveL Offs(pOrigin,144.27,162.46,0.00),v40,z0,tPen\WObj:=wPaper;
    MoveL Offs(pOrigin,144.44,161.40,0.00),v40,z0,tPen\WObj:=wPaper;
    MoveL Offs(pOrigin,144.44,161.40,0.00),v40,z0,tPen\WObj:=wPaper;
    MoveL Offs(pOrigin,145.26,159.91,0.00),v40,z0,tPen\WObj:=wPaper;
    MoveL Offs(pOrigin,144.98,159.24,0.00),v40,z0,tPen\WObj:=wPaper;
    MoveL Offs(pOrigin,143.17,160.69,0.00),v40,z0,tPen\WObj:=wPaper;
    MoveL Offs(pOrigin,142.32,160.98,0.00),v40,z0,tPen\WObj:=wPaper;
    MoveL Offs(pOrigin,140.62,160.87,0.00),v40,z0,tPen\WObj:=wPaper;
    MoveL Offs(pOrigin,138.39,159.70,0.00),v40,z0,tPen\WObj:=wPaper;
    MoveL Offs(pOrigin,138.39,159.70,0.00),v40,z0,tPen\WObj:=wPaper;
    MoveL Offs(pOrigin,139.45,159.70,0.00),v40,z0,tPen\WObj:=wPaper;
    MoveL Offs(pOrigin,138.39,159.70,0.00),v40,z0,tPen\WObj:=wPaper;
    MoveL Offs(pOrigin,135.52,158.96,0.00),v40,z0,tPen\WObj:=wPaper;
    MoveL Offs(pOrigin,135.52,158.96,0.00),v40,z0,tPen\WObj:=wPaper;
    MoveL Offs(pOrigin,134.07,159.38,0.00),v40,z0,tPen\WObj:=wPaper;
    MoveL Offs(pOrigin,134.67,160.12,0.00),v40,z0,tPen\WObj:=wPaper;
    MoveL Offs(pOrigin,134.67,160.12,0.00),v40,z0,tPen\WObj:=wPaper;
    MoveL Offs(pOrigin,133.61,160.23,0.00),v40,z0,tPen\WObj:=wPaper;
    MoveL Offs(pOrigin,133.07,160.66,0.00),v40,z0,tPen\WObj:=wPaper;
    MoveL Offs(pOrigin,133.07,160.66,0.00),v40,z0,tPen\WObj:=wPaper;
    MoveL Offs(pOrigin,133.39,161.05,0.00),v40,z0,tPen\WObj:=wPaper;
    MoveL Offs(pOrigin,134.46,161.19,0.00),v40,fine,tPen\WObj:=wPaper;
    MoveL Offs(pOrigin,134.46,161.19,6.00),v60,z5,tPen\WObj:=wPaper;
    MoveL Offs(pOrigin,135.31,160.23,6.00),vTravel,z5,tPen\WObj:=wPaper;
    MoveL Offs(pOrigin,135.31,160.23,0.00),v60,z0,tPen\WObj:=wPaper;
    MoveL Offs(pOrigin,137.01,160.41,0.00),v40,z0,tPen\WObj:=wPaper;
    MoveL Offs(pOrigin,140.30,162.36,0.00),v40,z0,tPen\WObj:=wPaper;
    MoveL Offs(pOrigin,143.06,162.25,0.00),v40,fine,tPen\WObj:=wPaper;
    MoveL Offs(pOrigin,143.06,162.25,6.00),v60,z5,tPen\WObj:=wPaper;
    MoveL Offs(pOrigin,144.44,161.40,6.00),vTravel,z5,tPen\WObj:=wPaper;
    MoveL Offs(pOrigin,144.44,161.40,0.00),v60,z0,tPen\WObj:=wPaper;
    MoveL Offs(pOrigin,141.89,163.42,0.00),v40,fine,tPen\WObj:=wPaper;
    MoveL Offs(pOrigin,141.89,163.42,6.00),v60,z5,tPen\WObj:=wPaper;
    MoveL Offs(pOrigin,137.43,166.39,6.00),vTravel,z5,tPen\WObj:=wPaper;
    MoveL Offs(pOrigin,137.43,166.39,0.00),v60,z0,tPen\WObj:=wPaper;
    MoveL Offs(pOrigin,135.94,165.76,0.00),v40,z0,tPen\WObj:=wPaper;
    MoveL Offs(pOrigin,135.94,165.76,0.00),v40,z0,tPen\WObj:=wPaper;
    MoveL Offs(pOrigin,133.18,162.78,0.00),v40,fine,tPen\WObj:=wPaper;
    MoveL Offs(pOrigin,133.18,162.78,6.00),v60,z5,tPen\WObj:=wPaper;
    MoveL Offs(pOrigin,131.69,162.04,6.00),vTravel,z5,tPen\WObj:=wPaper;
    MoveL Offs(pOrigin,131.69,162.04,0.00),v60,z0,tPen\WObj:=wPaper;
    MoveL Offs(pOrigin,129.89,161.33,0.00),v40,z0,tPen\WObj:=wPaper;
    MoveL Offs(pOrigin,129.68,160.98,0.00),v40,z0,tPen\WObj:=wPaper;
    MoveL Offs(pOrigin,129.68,160.98,0.00),v40,z0,tPen\WObj:=wPaper;
    MoveL Offs(pOrigin,130.42,160.76,0.00),v40,z0,tPen\WObj:=wPaper;
    MoveL Offs(pOrigin,131.48,160.98,0.00),v40,z0,tPen\WObj:=wPaper;
    MoveL Offs(pOrigin,132.01,160.55,0.00),v40,z0,tPen\WObj:=wPaper;
    MoveL Offs(pOrigin,132.01,160.55,0.00),v40,z0,tPen\WObj:=wPaper;
    MoveL Offs(pOrigin,133.07,160.66,0.00),v40,z0,tPen\WObj:=wPaper;
    MoveL Offs(pOrigin,132.01,160.55,0.00),v40,z0,tPen\WObj:=wPaper;
    MoveL Offs(pOrigin,129.57,159.52,0.00),v40,z0,tPen\WObj:=wPaper;
    MoveL Offs(pOrigin,128.08,158.11,0.00),v40,z0,tPen\WObj:=wPaper;
    MoveL Offs(pOrigin,126.91,158.11,0.00),v40,z0,tPen\WObj:=wPaper;
  ENDPROC

  PROC DrawPart16()
    MoveL Offs(pOrigin,127.12,159.17,0.00),v40,z0,tPen\WObj:=wPaper;
    MoveL Offs(pOrigin,127.12,159.17,0.00),v40,z0,tPen\WObj:=wPaper;
    MoveL Offs(pOrigin,126.70,159.06,0.00),v40,z0,tPen\WObj:=wPaper;
    MoveL Offs(pOrigin,126.38,158.32,0.00),v40,z0,tPen\WObj:=wPaper;
    MoveL Offs(pOrigin,126.06,158.74,0.00),v40,z0,tPen\WObj:=wPaper;
    MoveL Offs(pOrigin,126.17,160.02,0.00),v40,z0,tPen\WObj:=wPaper;
    MoveL Offs(pOrigin,126.17,160.02,0.00),v40,z0,tPen\WObj:=wPaper;
    MoveL Offs(pOrigin,125.71,159.70,0.00),v40,z0,tPen\WObj:=wPaper;
    MoveL Offs(pOrigin,125.53,158.43,0.00),v40,z0,tPen\WObj:=wPaper;
    MoveL Offs(pOrigin,124.79,158.53,0.00),v40,z0,tPen\WObj:=wPaper;
    MoveL Offs(pOrigin,124.57,159.38,0.00),v40,z0,tPen\WObj:=wPaper;
    MoveL Offs(pOrigin,124.93,160.44,0.00),v40,z0,tPen\WObj:=wPaper;
    MoveL Offs(pOrigin,125.74,161.51,0.00),v40,z0,tPen\WObj:=wPaper;
    MoveL Offs(pOrigin,126.38,161.72,0.00),v40,z0,tPen\WObj:=wPaper;
    MoveL Offs(pOrigin,126.38,161.72,0.00),v40,z0,tPen\WObj:=wPaper;
    MoveL Offs(pOrigin,128.08,163.10,0.00),v40,z0,tPen\WObj:=wPaper;
    MoveL Offs(pOrigin,128.51,163.84,0.00),v40,z0,tPen\WObj:=wPaper;
    MoveL Offs(pOrigin,128.51,163.84,0.00),v40,z0,tPen\WObj:=wPaper;
    MoveL Offs(pOrigin,127.02,163.63,0.00),v40,z0,tPen\WObj:=wPaper;
    MoveL Offs(pOrigin,127.02,163.63,0.00),v40,z0,tPen\WObj:=wPaper;
    MoveL Offs(pOrigin,128.08,166.18,0.00),v40,z0,tPen\WObj:=wPaper;
    MoveL Offs(pOrigin,127.69,168.09,0.00),v40,z0,tPen\WObj:=wPaper;
    MoveL Offs(pOrigin,126.91,169.26,0.00),v40,fine,tPen\WObj:=wPaper;
    MoveL Offs(pOrigin,126.91,169.26,6.00),v60,z5,tPen\WObj:=wPaper;
    MoveL Offs(pOrigin,127.02,170.64,6.00),vTravel,z5,tPen\WObj:=wPaper;
    MoveL Offs(pOrigin,127.02,170.64,0.00),v60,z0,tPen\WObj:=wPaper;
    MoveL Offs(pOrigin,128.40,168.52,0.00),v40,z0,tPen\WObj:=wPaper;
    MoveL Offs(pOrigin,129.14,169.05,0.00),v40,z0,tPen\WObj:=wPaper;
    MoveL Offs(pOrigin,129.36,166.18,0.00),v40,z0,tPen\WObj:=wPaper;
    MoveL Offs(pOrigin,129.04,164.48,0.00),v40,z0,tPen\WObj:=wPaper;
    MoveL Offs(pOrigin,129.04,164.48,0.00),v40,z0,tPen\WObj:=wPaper;
    MoveL Offs(pOrigin,129.64,164.80,0.00),v40,z0,tPen\WObj:=wPaper;
    MoveL Offs(pOrigin,130.10,165.86,0.00),v40,z0,tPen\WObj:=wPaper;
    MoveL Offs(pOrigin,130.10,168.09,0.00),v40,z0,tPen\WObj:=wPaper;
    MoveL Offs(pOrigin,129.82,168.73,0.00),v40,z0,tPen\WObj:=wPaper;
    MoveL Offs(pOrigin,126.88,171.71,0.00),v40,z0,tPen\WObj:=wPaper;
    MoveL Offs(pOrigin,127.87,171.71,0.00),v40,z0,tPen\WObj:=wPaper;
    MoveL Offs(pOrigin,129.57,170.96,0.00),v40,fine,tPen\WObj:=wPaper;
    MoveL Offs(pOrigin,129.57,170.96,6.00),v60,z5,tPen\WObj:=wPaper;
    MoveL Offs(pOrigin,131.48,170.54,6.00),vTravel,z5,tPen\WObj:=wPaper;
    MoveL Offs(pOrigin,131.48,170.54,0.00),v60,z0,tPen\WObj:=wPaper;
    MoveL Offs(pOrigin,132.76,170.32,0.00),v40,fine,tPen\WObj:=wPaper;
    MoveL Offs(pOrigin,132.76,170.32,6.00),v60,z5,tPen\WObj:=wPaper;
    MoveL Offs(pOrigin,134.67,167.99,6.00),vTravel,z5,tPen\WObj:=wPaper;
    MoveL Offs(pOrigin,134.67,167.99,0.00),v60,z0,tPen\WObj:=wPaper;
    MoveL Offs(pOrigin,135.62,167.46,0.00),v40,z0,tPen\WObj:=wPaper;
    MoveL Offs(pOrigin,135.94,166.61,0.00),v40,z0,tPen\WObj:=wPaper;
    MoveL Offs(pOrigin,135.94,166.61,0.00),v40,z0,tPen\WObj:=wPaper;
    MoveL Offs(pOrigin,135.73,165.90,0.00),v40,z0,tPen\WObj:=wPaper;
    MoveL Offs(pOrigin,134.81,165.76,0.00),v40,z0,tPen\WObj:=wPaper;
    MoveL Offs(pOrigin,134.67,167.99,0.00),v40,fine,tPen\WObj:=wPaper;
    MoveL Offs(pOrigin,134.67,167.99,6.00),v60,z5,tPen\WObj:=wPaper;
    MoveL Offs(pOrigin,135.94,166.61,6.00),vTravel,z5,tPen\WObj:=wPaper;
    MoveL Offs(pOrigin,135.94,166.61,0.00),v60,z0,tPen\WObj:=wPaper;
    MoveL Offs(pOrigin,137.01,166.82,0.00),v40,fine,tPen\WObj:=wPaper;
    MoveL Offs(pOrigin,137.01,166.82,6.00),v60,z5,tPen\WObj:=wPaper;
    MoveL Offs(pOrigin,130.63,163.84,6.00),vTravel,z5,tPen\WObj:=wPaper;
    MoveL Offs(pOrigin,130.63,163.84,0.00),v60,z0,tPen\WObj:=wPaper;
    MoveL Offs(pOrigin,130.95,164.16,0.00),v40,z0,tPen\WObj:=wPaper;
    MoveL Offs(pOrigin,130.63,163.84,0.00),v40,z0,tPen\WObj:=wPaper;
    MoveL Offs(pOrigin,130.10,163.31,0.00),v40,z0,tPen\WObj:=wPaper;
    MoveL Offs(pOrigin,130.52,163.74,0.00),v40,z0,tPen\WObj:=wPaper;
    MoveL Offs(pOrigin,130.10,163.31,0.00),v40,z0,tPen\WObj:=wPaper;
    MoveL Offs(pOrigin,129.78,162.78,0.00),v40,z0,tPen\WObj:=wPaper;
    MoveL Offs(pOrigin,127.97,161.51,0.00),v40,z0,tPen\WObj:=wPaper;
    MoveL Offs(pOrigin,127.97,161.51,0.00),v40,z0,tPen\WObj:=wPaper;
    MoveL Offs(pOrigin,127.66,160.98,0.00),v40,z0,tPen\WObj:=wPaper;
    MoveL Offs(pOrigin,127.12,160.87,0.00),v40,z0,tPen\WObj:=wPaper;
    MoveL Offs(pOrigin,126.49,160.66,0.00),v40,z0,tPen\WObj:=wPaper;
    MoveL Offs(pOrigin,127.76,161.72,0.00),v40,fine,tPen\WObj:=wPaper;
    MoveL Offs(pOrigin,127.76,161.72,6.00),v60,z5,tPen\WObj:=wPaper;
    MoveL Offs(pOrigin,129.68,160.98,6.00),vTravel,z5,tPen\WObj:=wPaper;
    MoveL Offs(pOrigin,129.68,160.98,0.00),v60,z0,tPen\WObj:=wPaper;
    MoveL Offs(pOrigin,128.19,160.23,0.00),v40,z0,tPen\WObj:=wPaper;
    MoveL Offs(pOrigin,127.12,159.17,0.00),v40,fine,tPen\WObj:=wPaper;
    MoveL Offs(pOrigin,127.12,159.17,6.00),v60,z5,tPen\WObj:=wPaper;
    MoveL Offs(pOrigin,123.51,158.43,6.00),vTravel,z5,tPen\WObj:=wPaper;
    MoveL Offs(pOrigin,123.51,158.43,0.00),v60,z0,tPen\WObj:=wPaper;
    MoveL Offs(pOrigin,123.65,160.44,0.00),v40,z0,tPen\WObj:=wPaper;
    MoveL Offs(pOrigin,124.89,162.25,0.00),v40,z0,tPen\WObj:=wPaper;
    MoveL Offs(pOrigin,124.89,162.25,0.00),v40,z0,tPen\WObj:=wPaper;
    MoveL Offs(pOrigin,123.41,161.72,0.00),v40,z0,tPen\WObj:=wPaper;
    MoveL Offs(pOrigin,122.98,162.14,0.00),v40,z0,tPen\WObj:=wPaper;
    MoveL Offs(pOrigin,122.98,162.14,0.00),v40,z0,tPen\WObj:=wPaper;
    MoveL Offs(pOrigin,122.03,161.82,0.00),v40,z0,tPen\WObj:=wPaper;
    MoveL Offs(pOrigin,121.07,160.80,0.00),v40,z0,tPen\WObj:=wPaper;
    MoveL Offs(pOrigin,121.28,162.04,0.00),v40,z0,tPen\WObj:=wPaper;
    MoveL Offs(pOrigin,121.07,162.36,0.00),v40,z0,tPen\WObj:=wPaper;
    MoveL Offs(pOrigin,121.07,162.36,0.00),v40,z0,tPen\WObj:=wPaper;
    MoveL Offs(pOrigin,120.01,161.29,0.00),v40,z0,tPen\WObj:=wPaper;
    MoveL Offs(pOrigin,119.47,160.02,0.00),v40,z0,tPen\WObj:=wPaper;
    MoveL Offs(pOrigin,119.47,158.85,0.00),v40,z0,tPen\WObj:=wPaper;
    MoveL Offs(pOrigin,120.11,157.57,0.00),v40,z0,tPen\WObj:=wPaper;
    MoveL Offs(pOrigin,119.05,157.68,0.00),v40,z0,tPen\WObj:=wPaper;
    MoveL Offs(pOrigin,118.41,159.27,0.00),v40,z0,tPen\WObj:=wPaper;
    MoveL Offs(pOrigin,118.73,161.51,0.00),v40,z0,tPen\WObj:=wPaper;
    MoveL Offs(pOrigin,118.73,161.51,0.00),v40,z0,tPen\WObj:=wPaper;
    MoveL Offs(pOrigin,119.16,162.46,0.00),v40,z0,tPen\WObj:=wPaper;
    MoveL Offs(pOrigin,120.96,164.06,0.00),v40,z0,tPen\WObj:=wPaper;
    MoveL Offs(pOrigin,121.18,164.06,0.00),v40,z0,tPen\WObj:=wPaper;
    MoveL Offs(pOrigin,122.34,164.38,0.00),v40,z0,tPen\WObj:=wPaper;
    MoveL Offs(pOrigin,122.88,164.91,0.00),v40,z0,tPen\WObj:=wPaper;
    MoveL Offs(pOrigin,123.62,166.93,0.00),v40,z0,tPen\WObj:=wPaper;
    MoveL Offs(pOrigin,123.23,168.73,0.00),v40,z0,tPen\WObj:=wPaper;
    MoveL Offs(pOrigin,121.49,170.32,0.00),v40,z0,tPen\WObj:=wPaper;
    MoveL Offs(pOrigin,121.42,169.79,0.00),v40,z0,tPen\WObj:=wPaper;
    MoveL Offs(pOrigin,122.34,168.31,0.00),v40,z0,tPen\WObj:=wPaper;
    MoveL Offs(pOrigin,122.45,166.82,0.00),v40,z0,tPen\WObj:=wPaper;
    MoveL Offs(pOrigin,121.03,164.27,0.00),v40,z0,tPen\WObj:=wPaper;
    MoveL Offs(pOrigin,121.18,164.06,0.00),v40,z0,tPen\WObj:=wPaper;
    MoveL Offs(pOrigin,121.49,163.31,0.00),v40,z0,tPen\WObj:=wPaper;
    MoveL Offs(pOrigin,121.92,163.74,0.00),v40,z0,tPen\WObj:=wPaper;
    MoveL Offs(pOrigin,121.49,163.31,0.00),v40,z0,tPen\WObj:=wPaper;
    MoveL Offs(pOrigin,121.39,162.57,0.00),v40,z0,tPen\WObj:=wPaper;
    MoveL Offs(pOrigin,121.21,162.99,0.00),v40,z0,tPen\WObj:=wPaper;
    MoveL Offs(pOrigin,122.24,164.27,0.00),v40,fine,tPen\WObj:=wPaper;
    MoveL Offs(pOrigin,122.24,164.27,6.00),v60,z5,tPen\WObj:=wPaper;
    MoveL Offs(pOrigin,121.39,162.57,6.00),vTravel,z5,tPen\WObj:=wPaper;
    MoveL Offs(pOrigin,121.39,162.57,0.00),v60,z0,tPen\WObj:=wPaper;
    MoveL Offs(pOrigin,124.15,164.30,0.00),v40,z0,tPen\WObj:=wPaper;
  ENDPROC

  PROC DrawPart17()
    MoveL Offs(pOrigin,124.82,165.44,0.00),v40,z0,tPen\WObj:=wPaper;
    MoveL Offs(pOrigin,125.21,167.46,0.00),v40,z0,tPen\WObj:=wPaper;
    MoveL Offs(pOrigin,124.36,169.86,0.00),v40,z0,tPen\WObj:=wPaper;
    MoveL Offs(pOrigin,125.64,168.94,0.00),v40,z0,tPen\WObj:=wPaper;
    MoveL Offs(pOrigin,126.49,167.24,0.00),v40,z0,tPen\WObj:=wPaper;
    MoveL Offs(pOrigin,126.42,165.33,0.00),v40,z0,tPen\WObj:=wPaper;
    MoveL Offs(pOrigin,125.74,164.16,0.00),v40,z0,tPen\WObj:=wPaper;
    MoveL Offs(pOrigin,125.21,163.88,0.00),v40,z0,tPen\WObj:=wPaper;
    MoveL Offs(pOrigin,125.64,165.12,0.00),v40,fine,tPen\WObj:=wPaper;
    MoveL Offs(pOrigin,125.64,165.12,6.00),v60,z5,tPen\WObj:=wPaper;
    MoveL Offs(pOrigin,125.11,163.84,6.00),vTravel,z5,tPen\WObj:=wPaper;
    MoveL Offs(pOrigin,125.11,163.84,0.00),v60,z0,tPen\WObj:=wPaper;
    MoveL Offs(pOrigin,122.98,162.14,0.00),v40,z0,tPen\WObj:=wPaper;
    MoveL Offs(pOrigin,122.98,161.72,0.00),v40,z0,tPen\WObj:=wPaper;
    MoveL Offs(pOrigin,122.24,160.02,0.00),v40,z0,tPen\WObj:=wPaper;
    MoveL Offs(pOrigin,122.24,158.96,0.00),v40,z0,tPen\WObj:=wPaper;
    MoveL Offs(pOrigin,122.66,158.00,0.00),v40,fine,tPen\WObj:=wPaper;
    MoveL Offs(pOrigin,122.66,158.00,6.00),v60,z5,tPen\WObj:=wPaper;
    MoveL Offs(pOrigin,120.86,158.96,6.00),vTravel,z5,tPen\WObj:=wPaper;
    MoveL Offs(pOrigin,120.86,158.96,0.00),v60,z0,tPen\WObj:=wPaper;
    MoveL Offs(pOrigin,120.96,160.76,0.00),v40,fine,tPen\WObj:=wPaper;
    MoveL Offs(pOrigin,120.96,160.76,6.00),v60,z5,tPen\WObj:=wPaper;
    MoveL Offs(pOrigin,118.73,161.51,6.00),vTravel,z5,tPen\WObj:=wPaper;
    MoveL Offs(pOrigin,118.73,161.51,0.00),v60,z0,tPen\WObj:=wPaper;
    MoveL Offs(pOrigin,118.09,161.19,0.00),v40,z0,tPen\WObj:=wPaper;
    MoveL Offs(pOrigin,117.56,160.02,0.00),v40,z0,tPen\WObj:=wPaper;
    MoveL Offs(pOrigin,117.56,158.85,0.00),v40,z0,tPen\WObj:=wPaper;
    MoveL Offs(pOrigin,118.41,157.36,0.00),v40,fine,tPen\WObj:=wPaper;
    MoveL Offs(pOrigin,118.41,157.36,6.00),v60,z5,tPen\WObj:=wPaper;
    MoveL Offs(pOrigin,116.93,157.79,6.00),vTravel,z5,tPen\WObj:=wPaper;
    MoveL Offs(pOrigin,116.93,157.79,0.00),v60,z0,tPen\WObj:=wPaper;
    MoveL Offs(pOrigin,116.50,160.02,0.00),v40,z0,tPen\WObj:=wPaper;
    MoveL Offs(pOrigin,117.67,162.57,0.00),v40,z0,tPen\WObj:=wPaper;
    MoveL Offs(pOrigin,117.67,162.57,0.00),v40,z0,tPen\WObj:=wPaper;
    MoveL Offs(pOrigin,118.20,163.42,0.00),v40,z0,tPen\WObj:=wPaper;
    MoveL Offs(pOrigin,118.20,163.42,0.00),v40,z0,tPen\WObj:=wPaper;
    MoveL Offs(pOrigin,117.14,163.52,0.00),v40,z0,tPen\WObj:=wPaper;
    MoveL Offs(pOrigin,117.14,163.52,0.00),v40,z0,tPen\WObj:=wPaper;
    MoveL Offs(pOrigin,118.73,166.29,0.00),v40,z0,tPen\WObj:=wPaper;
    MoveL Offs(pOrigin,118.55,167.77,0.00),v40,z0,tPen\WObj:=wPaper;
    MoveL Offs(pOrigin,117.88,168.84,0.00),v40,z0,tPen\WObj:=wPaper;
    MoveL Offs(pOrigin,117.67,168.94,0.00),v40,z0,tPen\WObj:=wPaper;
    MoveL Offs(pOrigin,116.18,170.22,0.00),v40,fine,tPen\WObj:=wPaper;
    MoveL Offs(pOrigin,116.18,170.22,6.00),v60,z5,tPen\WObj:=wPaper;
    MoveL Offs(pOrigin,115.76,172.24,6.00),vTravel,z5,tPen\WObj:=wPaper;
    MoveL Offs(pOrigin,115.76,172.24,0.00),v60,z0,tPen\WObj:=wPaper;
    MoveL Offs(pOrigin,116.29,171.81,0.00),v40,z0,tPen\WObj:=wPaper;
    MoveL Offs(pOrigin,118.41,171.64,0.00),v40,z0,tPen\WObj:=wPaper;
    MoveL Offs(pOrigin,121.28,170.32,0.00),v40,fine,tPen\WObj:=wPaper;
    MoveL Offs(pOrigin,121.28,170.32,6.00),v60,z5,tPen\WObj:=wPaper;
    MoveL Offs(pOrigin,120.64,172.02,6.00),vTravel,z5,tPen\WObj:=wPaper;
    MoveL Offs(pOrigin,120.64,172.02,0.00),v60,z0,tPen\WObj:=wPaper;
    MoveL Offs(pOrigin,120.96,171.56,0.00),v40,z0,tPen\WObj:=wPaper;
    MoveL Offs(pOrigin,124.26,169.90,0.00),v40,fine,tPen\WObj:=wPaper;
    MoveL Offs(pOrigin,124.26,169.90,6.00),v60,z5,tPen\WObj:=wPaper;
    MoveL Offs(pOrigin,124.79,171.92,6.00),vTravel,z5,tPen\WObj:=wPaper;
    MoveL Offs(pOrigin,124.79,171.92,0.00),v60,z0,tPen\WObj:=wPaper;
    MoveL Offs(pOrigin,115.86,172.34,0.00),v40,z0,tPen\WObj:=wPaper;
    MoveL Offs(pOrigin,112.89,171.81,0.00),v40,z0,tPen\WObj:=wPaper;
    MoveL Offs(pOrigin,109.06,170.47,0.00),v40,z0,tPen\WObj:=wPaper;
    MoveL Offs(pOrigin,108.53,170.01,0.00),v40,z0,tPen\WObj:=wPaper;
    MoveL Offs(pOrigin,106.09,169.62,0.00),v40,z0,tPen\WObj:=wPaper;
    MoveL Offs(pOrigin,105.88,169.26,0.00),v40,z0,tPen\WObj:=wPaper;
    MoveL Offs(pOrigin,105.88,169.26,0.00),v40,z0,tPen\WObj:=wPaper;
    MoveL Offs(pOrigin,107.47,168.84,0.00),v40,z0,tPen\WObj:=wPaper;
    MoveL Offs(pOrigin,107.47,168.84,0.00),v40,z0,tPen\WObj:=wPaper;
    MoveL Offs(pOrigin,111.51,169.30,0.00),v40,z0,tPen\WObj:=wPaper;
    MoveL Offs(pOrigin,113.63,168.84,0.00),v40,z0,tPen\WObj:=wPaper;
    MoveL Offs(pOrigin,113.63,168.84,0.00),v40,z0,tPen\WObj:=wPaper;
    MoveL Offs(pOrigin,113.53,167.99,0.00),v40,z0,tPen\WObj:=wPaper;
    MoveL Offs(pOrigin,111.29,168.20,0.00),v40,z0,tPen\WObj:=wPaper;
    MoveL Offs(pOrigin,110.87,167.99,0.00),v40,z0,tPen\WObj:=wPaper;
    MoveL Offs(pOrigin,110.87,167.99,0.00),v40,z0,tPen\WObj:=wPaper;
    MoveL Offs(pOrigin,111.93,167.35,0.00),v40,z0,tPen\WObj:=wPaper;
    MoveL Offs(pOrigin,111.93,167.35,0.00),v40,z0,tPen\WObj:=wPaper;
    MoveL Offs(pOrigin,113.53,166.50,0.00),v40,z0,tPen\WObj:=wPaper;
    MoveL Offs(pOrigin,114.06,165.44,0.00),v40,z0,tPen\WObj:=wPaper;
    MoveL Offs(pOrigin,113.77,163.84,0.00),v40,z0,tPen\WObj:=wPaper;
    MoveL Offs(pOrigin,112.14,161.51,0.00),v40,z0,tPen\WObj:=wPaper;
    MoveL Offs(pOrigin,112.14,161.51,0.00),v40,z0,tPen\WObj:=wPaper;
    MoveL Offs(pOrigin,112.57,160.44,0.00),v40,z0,tPen\WObj:=wPaper;
    MoveL Offs(pOrigin,113.21,160.55,0.00),v40,z0,tPen\WObj:=wPaper;
    MoveL Offs(pOrigin,113.74,161.72,0.00),v40,z0,tPen\WObj:=wPaper;
    MoveL Offs(pOrigin,114.48,162.14,0.00),v40,z0,tPen\WObj:=wPaper;
    MoveL Offs(pOrigin,114.48,162.14,0.00),v40,z0,tPen\WObj:=wPaper;
    MoveL Offs(pOrigin,114.59,161.08,0.00),v40,z0,tPen\WObj:=wPaper;
    MoveL Offs(pOrigin,114.59,161.08,0.00),v40,z0,tPen\WObj:=wPaper;
    MoveL Offs(pOrigin,114.06,160.44,0.00),v40,z0,tPen\WObj:=wPaper;
    MoveL Offs(pOrigin,114.06,159.38,0.00),v40,z0,tPen\WObj:=wPaper;
    MoveL Offs(pOrigin,114.69,158.00,0.00),v40,z0,tPen\WObj:=wPaper;
    MoveL Offs(pOrigin,115.33,158.21,0.00),v40,z0,tPen\WObj:=wPaper;
    MoveL Offs(pOrigin,114.91,160.44,0.00),v40,z0,tPen\WObj:=wPaper;
    MoveL Offs(pOrigin,115.44,160.55,0.00),v40,z0,tPen\WObj:=wPaper;
    MoveL Offs(pOrigin,116.07,157.79,0.00),v40,fine,tPen\WObj:=wPaper;
    MoveL Offs(pOrigin,116.07,157.79,6.00),v60,z5,tPen\WObj:=wPaper;
    MoveL Offs(pOrigin,114.06,157.57,6.00),vTravel,z5,tPen\WObj:=wPaper;
    MoveL Offs(pOrigin,114.06,157.57,0.00),v60,z0,tPen\WObj:=wPaper;
    MoveL Offs(pOrigin,113.03,158.96,0.00),v40,z0,tPen\WObj:=wPaper;
    MoveL Offs(pOrigin,113.21,160.55,0.00),v40,z0,tPen\WObj:=wPaper;
    MoveL Offs(pOrigin,113.21,160.55,0.00),v40,z0,tPen\WObj:=wPaper;
    MoveL Offs(pOrigin,112.57,160.23,0.00),v40,z0,tPen\WObj:=wPaper;
    MoveL Offs(pOrigin,112.71,159.27,0.00),v40,z0,tPen\WObj:=wPaper;
    MoveL Offs(pOrigin,112.99,159.17,0.00),v40,fine,tPen\WObj:=wPaper;
    MoveL Offs(pOrigin,112.99,159.17,6.00),v60,z5,tPen\WObj:=wPaper;
    MoveL Offs(pOrigin,112.57,157.68,6.00),vTravel,z5,tPen\WObj:=wPaper;
    MoveL Offs(pOrigin,112.57,157.68,0.00),v60,z0,tPen\WObj:=wPaper;
    MoveL Offs(pOrigin,111.19,158.53,0.00),v40,z0,tPen\WObj:=wPaper;
    MoveL Offs(pOrigin,111.19,158.53,0.00),v40,z0,tPen\WObj:=wPaper;
    MoveL Offs(pOrigin,111.08,160.55,0.00),v40,z0,tPen\WObj:=wPaper;
    MoveL Offs(pOrigin,111.08,160.55,0.00),v40,z0,tPen\WObj:=wPaper;
    MoveL Offs(pOrigin,111.93,161.51,0.00),v40,z0,tPen\WObj:=wPaper;
    MoveL Offs(pOrigin,112.36,161.82,0.00),v40,z0,tPen\WObj:=wPaper;
    MoveL Offs(pOrigin,111.93,161.61,0.00),v40,z0,tPen\WObj:=wPaper;
    MoveL Offs(pOrigin,111.82,162.14,0.00),v40,z0,tPen\WObj:=wPaper;
    MoveL Offs(pOrigin,112.68,164.16,0.00),v40,z0,tPen\WObj:=wPaper;
    MoveL Offs(pOrigin,112.78,165.65,0.00),v40,z0,tPen\WObj:=wPaper;
    MoveL Offs(pOrigin,111.93,167.35,0.00),v40,fine,tPen\WObj:=wPaper;
    MoveL Offs(pOrigin,111.93,167.35,6.00),v60,z5,tPen\WObj:=wPaper;
    MoveL Offs(pOrigin,110.87,167.99,6.00),vTravel,z5,tPen\WObj:=wPaper;
    MoveL Offs(pOrigin,110.87,167.99,0.00),v60,z0,tPen\WObj:=wPaper;
  ENDPROC

  PROC DrawPart18()
    MoveL Offs(pOrigin,108.21,168.09,0.00),v40,z0,tPen\WObj:=wPaper;
    MoveL Offs(pOrigin,104.95,167.35,0.00),v40,z0,tPen\WObj:=wPaper;
    MoveL Offs(pOrigin,105.88,168.16,0.00),v40,z0,tPen\WObj:=wPaper;
    MoveL Offs(pOrigin,107.47,168.84,0.00),v40,fine,tPen\WObj:=wPaper;
    MoveL Offs(pOrigin,107.47,168.84,6.00),v60,z5,tPen\WObj:=wPaper;
    MoveL Offs(pOrigin,105.88,169.26,6.00),vTravel,z5,tPen\WObj:=wPaper;
    MoveL Offs(pOrigin,105.88,169.26,0.00),v60,z0,tPen\WObj:=wPaper;
    MoveL Offs(pOrigin,104.07,168.41,0.00),v40,z0,tPen\WObj:=wPaper;
    MoveL Offs(pOrigin,102.69,167.14,0.00),v40,z0,tPen\WObj:=wPaper;
    MoveL Offs(pOrigin,101.24,165.01,0.00),v40,z0,tPen\WObj:=wPaper;
    MoveL Offs(pOrigin,101.31,164.27,0.00),v40,z0,tPen\WObj:=wPaper;
    MoveL Offs(pOrigin,101.31,164.27,0.00),v40,z0,tPen\WObj:=wPaper;
    MoveL Offs(pOrigin,100.56,163.31,0.00),v40,z0,tPen\WObj:=wPaper;
    MoveL Offs(pOrigin,100.56,163.31,0.00),v40,z0,tPen\WObj:=wPaper;
    MoveL Offs(pOrigin,101.09,163.10,0.00),v40,z0,tPen\WObj:=wPaper;
    MoveL Offs(pOrigin,103.86,163.63,0.00),v40,z0,tPen\WObj:=wPaper;
    MoveL Offs(pOrigin,106.09,162.43,0.00),v40,z0,tPen\WObj:=wPaper;
    MoveL Offs(pOrigin,106.19,163.10,0.00),v40,z0,tPen\WObj:=wPaper;
    MoveL Offs(pOrigin,106.30,162.36,0.00),v40,z0,tPen\WObj:=wPaper;
    MoveL Offs(pOrigin,106.19,161.44,0.00),v40,z0,tPen\WObj:=wPaper;
    MoveL Offs(pOrigin,104.60,162.50,0.00),v40,z0,tPen\WObj:=wPaper;
    MoveL Offs(pOrigin,102.79,162.78,0.00),v40,z0,tPen\WObj:=wPaper;
    MoveL Offs(pOrigin,100.35,161.61,0.00),v40,z0,tPen\WObj:=wPaper;
    MoveL Offs(pOrigin,99.93,160.66,0.00),v40,z0,tPen\WObj:=wPaper;
    MoveL Offs(pOrigin,99.93,160.66,0.00),v40,z0,tPen\WObj:=wPaper;
    MoveL Offs(pOrigin,99.39,159.91,0.00),v40,z0,tPen\WObj:=wPaper;
    MoveL Offs(pOrigin,99.39,159.91,0.00),v40,z0,tPen\WObj:=wPaper;
    MoveL Offs(pOrigin,99.71,159.63,0.00),v40,z0,tPen\WObj:=wPaper;
    MoveL Offs(pOrigin,101.84,159.91,0.00),v40,z0,tPen\WObj:=wPaper;
    MoveL Offs(pOrigin,103.22,159.52,0.00),v40,z0,tPen\WObj:=wPaper;
    MoveL Offs(pOrigin,106.94,157.15,0.00),v40,z0,tPen\WObj:=wPaper;
    MoveL Offs(pOrigin,106.94,157.15,0.00),v40,z0,tPen\WObj:=wPaper;
    MoveL Offs(pOrigin,108.11,157.26,0.00),v40,z0,tPen\WObj:=wPaper;
    MoveL Offs(pOrigin,108.11,157.26,0.00),v40,z0,tPen\WObj:=wPaper;
    MoveL Offs(pOrigin,107.47,158.04,0.00),v40,z0,tPen\WObj:=wPaper;
    MoveL Offs(pOrigin,106.51,158.25,0.00),v40,z0,tPen\WObj:=wPaper;
    MoveL Offs(pOrigin,105.45,159.59,0.00),v40,z0,tPen\WObj:=wPaper;
    MoveL Offs(pOrigin,105.24,159.70,0.00),v40,z0,tPen\WObj:=wPaper;
    MoveL Offs(pOrigin,102.37,160.98,0.00),v40,fine,tPen\WObj:=wPaper;
    MoveL Offs(pOrigin,102.37,160.98,6.00),v60,z5,tPen\WObj:=wPaper;
    MoveL Offs(pOrigin,99.93,160.66,6.00),vTravel,z5,tPen\WObj:=wPaper;
    MoveL Offs(pOrigin,99.93,160.66,0.00),v60,z0,tPen\WObj:=wPaper;
    MoveL Offs(pOrigin,103.11,161.40,0.00),v40,z0,tPen\WObj:=wPaper;
    MoveL Offs(pOrigin,105.88,160.34,0.00),v40,z0,tPen\WObj:=wPaper;
    MoveL Offs(pOrigin,106.41,161.40,0.00),v40,z0,tPen\WObj:=wPaper;
    MoveL Offs(pOrigin,107.04,159.17,0.00),v40,z0,tPen\WObj:=wPaper;
    MoveL Offs(pOrigin,107.04,159.17,0.00),v40,z0,tPen\WObj:=wPaper;
    MoveL Offs(pOrigin,108.64,158.04,0.00),v40,z0,tPen\WObj:=wPaper;
    MoveL Offs(pOrigin,109.38,158.00,0.00),v40,z0,tPen\WObj:=wPaper;
    MoveL Offs(pOrigin,109.38,158.00,0.00),v40,z0,tPen\WObj:=wPaper;
    MoveL Offs(pOrigin,109.17,158.96,0.00),v40,z0,tPen\WObj:=wPaper;
    MoveL Offs(pOrigin,109.17,158.96,0.00),v40,z0,tPen\WObj:=wPaper;
    MoveL Offs(pOrigin,108.28,159.27,0.00),v40,z0,tPen\WObj:=wPaper;
    MoveL Offs(pOrigin,107.68,160.66,0.00),v40,z0,tPen\WObj:=wPaper;
    MoveL Offs(pOrigin,107.29,163.52,0.00),v40,z0,tPen\WObj:=wPaper;
    MoveL Offs(pOrigin,106.30,164.27,0.00),v40,z0,tPen\WObj:=wPaper;
    MoveL Offs(pOrigin,106.09,164.38,0.00),v40,z0,tPen\WObj:=wPaper;
    MoveL Offs(pOrigin,104.81,164.80,0.00),v40,z0,tPen\WObj:=wPaper;
    MoveL Offs(pOrigin,103.32,164.69,0.00),v40,z0,tPen\WObj:=wPaper;
    MoveL Offs(pOrigin,102.90,165.01,0.00),v40,z0,tPen\WObj:=wPaper;
    MoveL Offs(pOrigin,102.90,165.01,0.00),v40,z0,tPen\WObj:=wPaper;
    MoveL Offs(pOrigin,101.31,164.27,0.00),v40,fine,tPen\WObj:=wPaper;
    MoveL Offs(pOrigin,101.31,164.27,6.00),v60,z5,tPen\WObj:=wPaper;
    MoveL Offs(pOrigin,100.56,163.31,6.00),vTravel,z5,tPen\WObj:=wPaper;
    MoveL Offs(pOrigin,100.56,163.31,0.00),v60,z0,tPen\WObj:=wPaper;
    MoveL Offs(pOrigin,98.40,161.08,0.00),v40,z0,tPen\WObj:=wPaper;
    MoveL Offs(pOrigin,97.73,159.59,0.00),v40,z0,tPen\WObj:=wPaper;
    MoveL Offs(pOrigin,98.01,159.17,0.00),v40,z0,tPen\WObj:=wPaper;
    MoveL Offs(pOrigin,98.01,159.17,0.00),v40,z0,tPen\WObj:=wPaper;
    MoveL Offs(pOrigin,99.39,159.91,0.00),v40,fine,tPen\WObj:=wPaper;
    MoveL Offs(pOrigin,99.39,159.91,6.00),v60,z5,tPen\WObj:=wPaper;
    MoveL Offs(pOrigin,98.01,159.17,6.00),vTravel,z5,tPen\WObj:=wPaper;
    MoveL Offs(pOrigin,98.01,159.17,0.00),v60,z0,tPen\WObj:=wPaper;
    MoveL Offs(pOrigin,96.91,157.26,0.00),v40,z0,tPen\WObj:=wPaper;
    MoveL Offs(pOrigin,96.74,156.30,0.00),v40,z0,tPen\WObj:=wPaper;
    MoveL Offs(pOrigin,96.74,156.30,0.00),v40,z0,tPen\WObj:=wPaper;
    MoveL Offs(pOrigin,95.21,153.11,0.00),v40,z0,tPen\WObj:=wPaper;
    MoveL Offs(pOrigin,94.82,151.52,0.00),v40,z0,tPen\WObj:=wPaper;
    MoveL Offs(pOrigin,95.43,148.76,0.00),v40,z0,tPen\WObj:=wPaper;
    MoveL Offs(pOrigin,96.21,148.01,0.00),v40,z0,tPen\WObj:=wPaper;
    MoveL Offs(pOrigin,96.21,148.01,0.00),v40,z0,tPen\WObj:=wPaper;
    MoveL Offs(pOrigin,96.31,147.80,0.00),v40,z0,tPen\WObj:=wPaper;
    MoveL Offs(pOrigin,96.95,148.23,0.00),v40,z0,tPen\WObj:=wPaper;
    MoveL Offs(pOrigin,96.95,148.23,0.00),v40,z0,tPen\WObj:=wPaper;
    MoveL Offs(pOrigin,96.38,148.65,0.00),v40,z0,tPen\WObj:=wPaper;
    MoveL Offs(pOrigin,96.63,150.03,0.00),v40,z0,tPen\WObj:=wPaper;
    MoveL Offs(pOrigin,96.63,150.03,0.00),v40,z0,tPen\WObj:=wPaper;
    MoveL Offs(pOrigin,98.97,153.61,0.00),v40,z0,tPen\WObj:=wPaper;
    MoveL Offs(pOrigin,102.05,155.02,0.00),v40,z0,tPen\WObj:=wPaper;
    MoveL Offs(pOrigin,103.86,154.81,0.00),v40,z0,tPen\WObj:=wPaper;
    MoveL Offs(pOrigin,103.86,154.81,0.00),v40,z0,tPen\WObj:=wPaper;
    MoveL Offs(pOrigin,103.64,153.43,0.00),v40,z0,tPen\WObj:=wPaper;
    MoveL Offs(pOrigin,103.64,153.43,0.00),v40,z0,tPen\WObj:=wPaper;
    MoveL Offs(pOrigin,106.72,154.28,0.00),v40,z0,tPen\WObj:=wPaper;
    MoveL Offs(pOrigin,107.36,155.02,0.00),v40,z0,tPen\WObj:=wPaper;
    MoveL Offs(pOrigin,104.71,154.60,0.00),v40,z0,tPen\WObj:=wPaper;
    MoveL Offs(pOrigin,104.07,154.81,0.00),v40,z0,tPen\WObj:=wPaper;
    MoveL Offs(pOrigin,104.07,154.81,0.00),v40,z0,tPen\WObj:=wPaper;
    MoveL Offs(pOrigin,104.60,156.16,0.00),v40,z0,tPen\WObj:=wPaper;
    MoveL Offs(pOrigin,102.16,155.98,0.00),v40,z0,tPen\WObj:=wPaper;
    MoveL Offs(pOrigin,100.46,155.45,0.00),v40,fine,tPen\WObj:=wPaper;
    MoveL Offs(pOrigin,100.46,155.45,6.00),v60,z5,tPen\WObj:=wPaper;
    MoveL Offs(pOrigin,100.46,153.54,6.00),vTravel,z5,tPen\WObj:=wPaper;
    MoveL Offs(pOrigin,100.46,153.54,0.00),v60,z0,tPen\WObj:=wPaper;
    MoveL Offs(pOrigin,102.90,154.71,0.00),v40,fine,tPen\WObj:=wPaper;
    MoveL Offs(pOrigin,102.90,154.71,6.00),v60,z5,tPen\WObj:=wPaper;
    MoveL Offs(pOrigin,103.11,153.22,6.00),vTravel,z5,tPen\WObj:=wPaper;
    MoveL Offs(pOrigin,103.11,153.22,0.00),v60,z0,tPen\WObj:=wPaper;
    MoveL Offs(pOrigin,101.84,153.25,0.00),v40,z0,tPen\WObj:=wPaper;
    MoveL Offs(pOrigin,99.61,151.94,0.00),v40,z0,tPen\WObj:=wPaper;
    MoveL Offs(pOrigin,98.65,150.99,0.00),v40,z0,tPen\WObj:=wPaper;
    MoveL Offs(pOrigin,96.95,148.23,0.00),v40,z0,tPen\WObj:=wPaper;
    MoveL Offs(pOrigin,96.21,147.80,0.00),v40,z0,tPen\WObj:=wPaper;
    MoveL Offs(pOrigin,95.89,145.68,0.00),v40,z0,tPen\WObj:=wPaper;
    MoveL Offs(pOrigin,95.89,145.68,0.00),v40,z0,tPen\WObj:=wPaper;
    MoveL Offs(pOrigin,95.89,143.76,0.00),v40,z0,tPen\WObj:=wPaper;
    MoveL Offs(pOrigin,96.53,143.12,0.00),v40,z0,tPen\WObj:=wPaper;
    MoveL Offs(pOrigin,96.53,143.12,0.00),v40,z0,tPen\WObj:=wPaper;
    MoveL Offs(pOrigin,97.16,144.29,0.00),v40,z0,tPen\WObj:=wPaper;
    MoveL Offs(pOrigin,97.16,144.29,0.00),v40,z0,tPen\WObj:=wPaper;
  ENDPROC

  PROC DrawPart19()
    MoveL Offs(pOrigin,99.29,145.25,0.00),v40,z0,tPen\WObj:=wPaper;
    MoveL Offs(pOrigin,99.29,145.25,0.00),v40,z0,tPen\WObj:=wPaper;
    MoveL Offs(pOrigin,100.74,147.91,0.00),v40,z0,tPen\WObj:=wPaper;
    MoveL Offs(pOrigin,102.90,150.77,0.00),v40,z0,tPen\WObj:=wPaper;
    MoveL Offs(pOrigin,102.90,150.77,0.00),v40,z0,tPen\WObj:=wPaper;
    MoveL Offs(pOrigin,103.64,150.81,0.00),v40,z0,tPen\WObj:=wPaper;
    MoveL Offs(pOrigin,104.92,151.73,0.00),v40,fine,tPen\WObj:=wPaper;
    MoveL Offs(pOrigin,104.92,151.73,6.00),v60,z5,tPen\WObj:=wPaper;
    MoveL Offs(pOrigin,105.66,153.11,6.00),vTravel,z5,tPen\WObj:=wPaper;
    MoveL Offs(pOrigin,105.66,153.11,0.00),v60,z0,tPen\WObj:=wPaper;
    MoveL Offs(pOrigin,103.43,152.01,0.00),v40,z0,tPen\WObj:=wPaper;
    MoveL Offs(pOrigin,103.01,152.69,0.00),v40,z0,tPen\WObj:=wPaper;
    MoveL Offs(pOrigin,102.79,152.69,0.00),v40,z0,tPen\WObj:=wPaper;
    MoveL Offs(pOrigin,101.20,151.84,0.00),v40,z0,tPen\WObj:=wPaper;
    MoveL Offs(pOrigin,100.42,150.99,0.00),v40,z0,tPen\WObj:=wPaper;
    MoveL Offs(pOrigin,101.73,150.88,0.00),v40,z0,tPen\WObj:=wPaper;
    MoveL Offs(pOrigin,101.73,150.88,0.00),v40,z0,tPen\WObj:=wPaper;
    MoveL Offs(pOrigin,102.79,151.09,0.00),v40,z0,tPen\WObj:=wPaper;
    MoveL Offs(pOrigin,102.79,151.09,0.00),v40,z0,tPen\WObj:=wPaper;
    MoveL Offs(pOrigin,103.22,151.94,0.00),v40,fine,tPen\WObj:=wPaper;
    MoveL Offs(pOrigin,103.22,151.94,6.00),v60,z5,tPen\WObj:=wPaper;
    MoveL Offs(pOrigin,104.07,150.35,6.00),vTravel,z5,tPen\WObj:=wPaper;
    MoveL Offs(pOrigin,104.07,150.35,0.00),v60,z0,tPen\WObj:=wPaper;
    MoveL Offs(pOrigin,102.37,148.33,0.00),v40,z0,tPen\WObj:=wPaper;
    MoveL Offs(pOrigin,102.26,147.69,0.00),v40,z0,tPen\WObj:=wPaper;
    MoveL Offs(pOrigin,102.47,147.59,0.00),v40,z0,tPen\WObj:=wPaper;
    MoveL Offs(pOrigin,103.43,148.86,0.00),v40,fine,tPen\WObj:=wPaper;
    MoveL Offs(pOrigin,103.43,148.86,6.00),v60,z5,tPen\WObj:=wPaper;
    MoveL Offs(pOrigin,103.11,147.27,6.00),vTravel,z5,tPen\WObj:=wPaper;
    MoveL Offs(pOrigin,103.11,147.27,0.00),v60,z0,tPen\WObj:=wPaper;
    MoveL Offs(pOrigin,102.23,145.36,0.00),v40,z0,tPen\WObj:=wPaper;
    MoveL Offs(pOrigin,101.62,145.04,0.00),v40,z0,tPen\WObj:=wPaper;
    MoveL Offs(pOrigin,101.62,145.04,0.00),v40,z0,tPen\WObj:=wPaper;
    MoveL Offs(pOrigin,101.73,144.33,0.00),v40,z0,tPen\WObj:=wPaper;
    MoveL Offs(pOrigin,102.47,144.72,0.00),v40,z0,tPen\WObj:=wPaper;
    MoveL Offs(pOrigin,102.47,143.87,0.00),v40,z0,tPen\WObj:=wPaper;
    MoveL Offs(pOrigin,101.62,142.38,0.00),v40,z0,tPen\WObj:=wPaper;
    MoveL Offs(pOrigin,101.62,142.38,0.00),v40,z0,tPen\WObj:=wPaper;
    MoveL Offs(pOrigin,100.67,140.04,0.00),v40,z0,tPen\WObj:=wPaper;
    MoveL Offs(pOrigin,100.67,140.04,0.00),v40,z0,tPen\WObj:=wPaper;
    MoveL Offs(pOrigin,99.29,139.09,0.00),v40,z0,tPen\WObj:=wPaper;
    MoveL Offs(pOrigin,99.29,139.09,0.00),v40,z0,tPen\WObj:=wPaper;
    MoveL Offs(pOrigin,98.97,137.81,0.00),v40,z0,tPen\WObj:=wPaper;
    MoveL Offs(pOrigin,99.50,137.18,0.00),v40,z0,tPen\WObj:=wPaper;
    MoveL Offs(pOrigin,99.50,137.18,0.00),v40,z0,tPen\WObj:=wPaper;
    MoveL Offs(pOrigin,100.24,138.13,0.00),v40,z0,tPen\WObj:=wPaper;
    MoveL Offs(pOrigin,100.24,138.13,0.00),v40,z0,tPen\WObj:=wPaper;
    MoveL Offs(pOrigin,100.67,140.04,0.00),v40,fine,tPen\WObj:=wPaper;
    MoveL Offs(pOrigin,100.67,140.04,6.00),v60,z5,tPen\WObj:=wPaper;
    MoveL Offs(pOrigin,101.94,139.41,6.00),vTravel,z5,tPen\WObj:=wPaper;
    MoveL Offs(pOrigin,101.94,139.41,0.00),v60,z0,tPen\WObj:=wPaper;
    MoveL Offs(pOrigin,101.06,136.96,0.00),v40,z0,tPen\WObj:=wPaper;
    MoveL Offs(pOrigin,99.93,136.32,0.00),v40,z0,tPen\WObj:=wPaper;
    MoveL Offs(pOrigin,99.71,136.75,0.00),v40,z0,tPen\WObj:=wPaper;
    MoveL Offs(pOrigin,100.42,137.60,0.00),v40,z0,tPen\WObj:=wPaper;
    MoveL Offs(pOrigin,100.24,138.13,0.00),v40,fine,tPen\WObj:=wPaper;
    MoveL Offs(pOrigin,100.24,138.13,6.00),v60,z5,tPen\WObj:=wPaper;
    MoveL Offs(pOrigin,98.97,138.02,6.00),vTravel,z5,tPen\WObj:=wPaper;
    MoveL Offs(pOrigin,98.97,138.02,0.00),v60,z0,tPen\WObj:=wPaper;
    MoveL Offs(pOrigin,98.44,138.24,0.00),v40,z0,tPen\WObj:=wPaper;
    MoveL Offs(pOrigin,98.22,139.37,0.00),v40,z0,tPen\WObj:=wPaper;
    MoveL Offs(pOrigin,97.69,139.62,0.00),v40,z0,tPen\WObj:=wPaper;
    MoveL Offs(pOrigin,97.48,140.15,0.00),v40,z0,tPen\WObj:=wPaper;
    MoveL Offs(pOrigin,98.33,140.36,0.00),v40,z0,tPen\WObj:=wPaper;
    MoveL Offs(pOrigin,98.33,140.36,0.00),v40,z0,tPen\WObj:=wPaper;
    MoveL Offs(pOrigin,99.68,141.64,0.00),v40,z0,tPen\WObj:=wPaper;
    MoveL Offs(pOrigin,101.62,144.29,0.00),v40,z0,tPen\WObj:=wPaper;
    MoveL Offs(pOrigin,101.41,143.87,0.00),v40,z0,tPen\WObj:=wPaper;
    MoveL Offs(pOrigin,101.62,142.38,0.00),v40,z0,tPen\WObj:=wPaper;
    MoveL Offs(pOrigin,102.69,142.27,0.00),v40,z0,tPen\WObj:=wPaper;
    MoveL Offs(pOrigin,101.84,140.15,0.00),v40,z0,tPen\WObj:=wPaper;
    MoveL Offs(pOrigin,101.94,139.41,0.00),v40,z0,tPen\WObj:=wPaper;
    MoveL Offs(pOrigin,101.94,139.41,0.00),v40,z0,tPen\WObj:=wPaper;
    MoveL Offs(pOrigin,102.69,140.68,0.00),v40,fine,tPen\WObj:=wPaper;
    MoveL Offs(pOrigin,102.69,140.68,6.00),v60,z5,tPen\WObj:=wPaper;
    MoveL Offs(pOrigin,102.69,139.19,6.00),vTravel,z5,tPen\WObj:=wPaper;
    MoveL Offs(pOrigin,102.69,139.19,0.00),v60,z0,tPen\WObj:=wPaper;
    MoveL Offs(pOrigin,102.37,135.26,0.00),v40,z0,tPen\WObj:=wPaper;
    MoveL Offs(pOrigin,102.37,135.26,0.00),v40,z0,tPen\WObj:=wPaper;
    MoveL Offs(pOrigin,102.90,134.84,0.00),v40,z0,tPen\WObj:=wPaper;
    MoveL Offs(pOrigin,104.07,135.16,0.00),v40,fine,tPen\WObj:=wPaper;
    MoveL Offs(pOrigin,104.07,135.16,6.00),v60,z5,tPen\WObj:=wPaper;
    MoveL Offs(pOrigin,101.62,135.48,6.00),vTravel,z5,tPen\WObj:=wPaper;
    MoveL Offs(pOrigin,101.62,135.48,0.00),v60,z0,tPen\WObj:=wPaper;
    MoveL Offs(pOrigin,100.46,135.51,0.00),v40,z0,tPen\WObj:=wPaper;
    MoveL Offs(pOrigin,101.09,136.11,0.00),v40,fine,tPen\WObj:=wPaper;
    MoveL Offs(pOrigin,101.09,136.11,6.00),v60,z5,tPen\WObj:=wPaper;
    MoveL Offs(pOrigin,102.58,132.18,6.00),vTravel,z5,tPen\WObj:=wPaper;
    MoveL Offs(pOrigin,102.58,132.18,0.00),v60,z0,tPen\WObj:=wPaper;
    MoveL Offs(pOrigin,103.54,132.18,0.00),v40,fine,tPen\WObj:=wPaper;
    MoveL Offs(pOrigin,103.54,132.18,6.00),v60,z5,tPen\WObj:=wPaper;
    MoveL Offs(pOrigin,102.58,131.44,6.00),vTravel,z5,tPen\WObj:=wPaper;
    MoveL Offs(pOrigin,102.58,131.44,0.00),v60,z0,tPen\WObj:=wPaper;
    MoveL Offs(pOrigin,103.43,126.23,0.00),v40,z0,tPen\WObj:=wPaper;
    MoveL Offs(pOrigin,103.11,123.75,0.00),v40,z0,tPen\WObj:=wPaper;
    MoveL Offs(pOrigin,102.47,124.74,0.00),v40,z0,tPen\WObj:=wPaper;
    MoveL Offs(pOrigin,102.58,126.44,0.00),v40,fine,tPen\WObj:=wPaper;
    MoveL Offs(pOrigin,102.58,126.44,6.00),v60,z5,tPen\WObj:=wPaper;
    MoveL Offs(pOrigin,100.88,122.30,6.00),vTravel,z5,tPen\WObj:=wPaper;
    MoveL Offs(pOrigin,100.88,122.30,0.00),v60,z0,tPen\WObj:=wPaper;
    MoveL Offs(pOrigin,101.41,119.22,0.00),v40,z0,tPen\WObj:=wPaper;
    MoveL Offs(pOrigin,101.41,119.22,0.00),v40,z0,tPen\WObj:=wPaper;
    MoveL Offs(pOrigin,102.26,116.88,0.00),v40,z0,tPen\WObj:=wPaper;
    MoveL Offs(pOrigin,103.11,116.35,0.00),v40,z0,tPen\WObj:=wPaper;
    MoveL Offs(pOrigin,104.18,116.35,0.00),v40,fine,tPen\WObj:=wPaper;
    MoveL Offs(pOrigin,104.18,116.35,6.00),v60,z5,tPen\WObj:=wPaper;
    MoveL Offs(pOrigin,101.41,119.22,6.00),vTravel,z5,tPen\WObj:=wPaper;
    MoveL Offs(pOrigin,101.41,119.22,0.00),v60,z0,tPen\WObj:=wPaper;
    MoveL Offs(pOrigin,95.25,117.77,0.00),v40,z0,tPen\WObj:=wPaper;
    MoveL Offs(pOrigin,91.00,115.75,0.00),v40,z0,tPen\WObj:=wPaper;
    MoveL Offs(pOrigin,87.92,112.95,0.00),v40,z0,tPen\WObj:=wPaper;
    MoveL Offs(pOrigin,86.64,110.19,0.00),v40,fine,tPen\WObj:=wPaper;
    MoveL Offs(pOrigin,86.64,110.19,6.00),v60,z5,tPen\WObj:=wPaper;
    MoveL Offs(pOrigin,99.07,100.62,6.00),vTravel,z5,tPen\WObj:=wPaper;
    MoveL Offs(pOrigin,99.07,100.62,0.00),v60,z0,tPen\WObj:=wPaper;
    MoveL Offs(pOrigin,99.50,101.05,0.00),v40,z0,tPen\WObj:=wPaper;
    MoveL Offs(pOrigin,99.07,100.62,0.00),v40,fine,tPen\WObj:=wPaper;
    MoveL Offs(pOrigin,99.07,100.62,6.00),v60,z5,tPen\WObj:=wPaper;
    MoveL Offs(pOrigin,106.41,131.76,6.00),vTravel,z5,tPen\WObj:=wPaper;
    MoveL Offs(pOrigin,106.41,131.76,0.00),v60,z0,tPen\WObj:=wPaper;
  ENDPROC

  PROC DrawPart20()
    MoveL Offs(pOrigin,108.11,132.04,0.00),v40,z0,tPen\WObj:=wPaper;
    MoveL Offs(pOrigin,108.74,132.71,0.00),v40,z0,tPen\WObj:=wPaper;
    MoveL Offs(pOrigin,108.74,132.71,0.00),v40,z0,tPen\WObj:=wPaper;
    MoveL Offs(pOrigin,110.02,133.14,0.00),v40,z0,tPen\WObj:=wPaper;
    MoveL Offs(pOrigin,110.02,133.14,0.00),v40,z0,tPen\WObj:=wPaper;
    MoveL Offs(pOrigin,110.12,133.56,0.00),v40,z0,tPen\WObj:=wPaper;
    MoveL Offs(pOrigin,111.08,134.27,0.00),v40,z0,tPen\WObj:=wPaper;
    MoveL Offs(pOrigin,111.82,134.31,0.00),v40,z0,tPen\WObj:=wPaper;
    MoveL Offs(pOrigin,111.82,134.31,0.00),v40,z0,tPen\WObj:=wPaper;
    MoveL Offs(pOrigin,111.97,133.77,0.00),v40,z0,tPen\WObj:=wPaper;
    MoveL Offs(pOrigin,112.68,133.35,0.00),v40,z0,tPen\WObj:=wPaper;
    MoveL Offs(pOrigin,112.68,133.35,0.00),v40,z0,tPen\WObj:=wPaper;
    MoveL Offs(pOrigin,111.93,132.61,0.00),v40,z0,tPen\WObj:=wPaper;
    MoveL Offs(pOrigin,110.02,133.14,0.00),v40,fine,tPen\WObj:=wPaper;
    MoveL Offs(pOrigin,110.02,133.14,6.00),v60,z5,tPen\WObj:=wPaper;
    MoveL Offs(pOrigin,108.74,132.71,6.00),vTravel,z5,tPen\WObj:=wPaper;
    MoveL Offs(pOrigin,108.74,132.71,0.00),v60,z0,tPen\WObj:=wPaper;
    MoveL Offs(pOrigin,109.06,133.67,0.00),v40,z0,tPen\WObj:=wPaper;
    MoveL Offs(pOrigin,109.91,134.41,0.00),v40,z0,tPen\WObj:=wPaper;
    MoveL Offs(pOrigin,112.57,135.48,0.00),v40,z0,tPen\WObj:=wPaper;
    MoveL Offs(pOrigin,115.01,135.58,0.00),v40,z0,tPen\WObj:=wPaper;
    MoveL Offs(pOrigin,117.03,134.62,0.00),v40,z0,tPen\WObj:=wPaper;
    MoveL Offs(pOrigin,117.67,134.73,0.00),v40,z0,tPen\WObj:=wPaper;
    MoveL Offs(pOrigin,117.67,134.73,0.00),v40,z0,tPen\WObj:=wPaper;
    MoveL Offs(pOrigin,117.60,135.69,0.00),v40,z0,tPen\WObj:=wPaper;
    MoveL Offs(pOrigin,116.82,136.36,0.00),v40,z0,tPen\WObj:=wPaper;
    MoveL Offs(pOrigin,115.44,136.64,0.00),v40,z0,tPen\WObj:=wPaper;
    MoveL Offs(pOrigin,109.70,136.22,0.00),v40,z0,tPen\WObj:=wPaper;
    MoveL Offs(pOrigin,107.79,135.62,0.00),v40,z0,tPen\WObj:=wPaper;
    MoveL Offs(pOrigin,106.72,134.62,0.00),v40,z0,tPen\WObj:=wPaper;
    MoveL Offs(pOrigin,106.51,133.88,0.00),v40,fine,tPen\WObj:=wPaper;
    MoveL Offs(pOrigin,106.51,133.88,6.00),v60,z5,tPen\WObj:=wPaper;
    MoveL Offs(pOrigin,111.82,134.31,6.00),vTravel,z5,tPen\WObj:=wPaper;
    MoveL Offs(pOrigin,111.82,134.31,0.00),v60,z0,tPen\WObj:=wPaper;
    MoveL Offs(pOrigin,112.46,134.73,0.00),v40,z0,tPen\WObj:=wPaper;
    MoveL Offs(pOrigin,113.21,134.62,0.00),v40,z0,tPen\WObj:=wPaper;
    MoveL Offs(pOrigin,113.21,134.62,0.00),v40,z0,tPen\WObj:=wPaper;
    MoveL Offs(pOrigin,113.17,133.56,0.00),v40,z0,tPen\WObj:=wPaper;
    MoveL Offs(pOrigin,112.68,133.35,0.00),v40,z0,tPen\WObj:=wPaper;
    MoveL Offs(pOrigin,112.14,132.61,0.00),v40,z0,tPen\WObj:=wPaper;
    MoveL Offs(pOrigin,112.46,132.93,0.00),v40,z0,tPen\WObj:=wPaper;
    MoveL Offs(pOrigin,112.14,132.61,0.00),v40,fine,tPen\WObj:=wPaper;
    MoveL Offs(pOrigin,112.14,132.61,6.00),v60,z5,tPen\WObj:=wPaper;
    MoveL Offs(pOrigin,111.93,130.80,6.00),vTravel,z5,tPen\WObj:=wPaper;
    MoveL Offs(pOrigin,111.93,130.80,0.00),v60,z0,tPen\WObj:=wPaper;
    MoveL Offs(pOrigin,116.39,132.18,0.00),v40,z0,tPen\WObj:=wPaper;
    MoveL Offs(pOrigin,117.35,132.50,0.00),v40,z0,tPen\WObj:=wPaper;
    MoveL Offs(pOrigin,117.99,133.67,0.00),v40,z0,tPen\WObj:=wPaper;
    MoveL Offs(pOrigin,117.67,134.62,0.00),v40,fine,tPen\WObj:=wPaper;
    MoveL Offs(pOrigin,117.67,134.62,6.00),v60,z5,tPen\WObj:=wPaper;
    MoveL Offs(pOrigin,118.84,133.56,6.00),vTravel,z5,tPen\WObj:=wPaper;
    MoveL Offs(pOrigin,118.84,133.56,0.00),v60,z0,tPen\WObj:=wPaper;
    MoveL Offs(pOrigin,118.52,133.24,0.00),v40,z0,tPen\WObj:=wPaper;
    MoveL Offs(pOrigin,118.73,132.61,0.00),v40,fine,tPen\WObj:=wPaper;
    MoveL Offs(pOrigin,118.73,132.61,6.00),v60,z5,tPen\WObj:=wPaper;
    MoveL Offs(pOrigin,117.35,132.50,6.00),vTravel,z5,tPen\WObj:=wPaper;
    MoveL Offs(pOrigin,117.35,132.50,0.00),v60,z0,tPen\WObj:=wPaper;
    MoveL Offs(pOrigin,114.48,130.06,0.00),v40,fine,tPen\WObj:=wPaper;
    MoveL Offs(pOrigin,114.48,130.06,6.00),v60,z5,tPen\WObj:=wPaper;
    MoveL Offs(pOrigin,113.84,133.56,6.00),vTravel,z5,tPen\WObj:=wPaper;
    MoveL Offs(pOrigin,113.84,133.56,0.00),v60,z0,tPen\WObj:=wPaper;
    MoveL Offs(pOrigin,114.27,133.99,0.00),v40,z0,tPen\WObj:=wPaper;
    MoveL Offs(pOrigin,114.27,134.62,0.00),v40,z0,tPen\WObj:=wPaper;
    MoveL Offs(pOrigin,114.27,134.62,0.00),v40,z0,tPen\WObj:=wPaper;
    MoveL Offs(pOrigin,116.18,133.88,0.00),v40,z0,tPen\WObj:=wPaper;
    MoveL Offs(pOrigin,116.18,133.88,0.00),v40,z0,tPen\WObj:=wPaper;
    MoveL Offs(pOrigin,115.97,133.42,0.00),v40,z0,tPen\WObj:=wPaper;
    MoveL Offs(pOrigin,114.48,133.03,0.00),v40,z0,tPen\WObj:=wPaper;
    MoveL Offs(pOrigin,113.84,133.56,0.00),v40,z0,tPen\WObj:=wPaper;
    MoveL Offs(pOrigin,114.27,134.62,0.00),v40,z0,tPen\WObj:=wPaper;
    MoveL Offs(pOrigin,113.21,134.62,0.00),v40,fine,tPen\WObj:=wPaper;
    MoveL Offs(pOrigin,113.21,134.62,6.00),v60,z5,tPen\WObj:=wPaper;
    MoveL Offs(pOrigin,116.18,133.88,6.00),vTravel,z5,tPen\WObj:=wPaper;
    MoveL Offs(pOrigin,116.18,133.88,0.00),v60,z0,tPen\WObj:=wPaper;
    MoveL Offs(pOrigin,117.03,133.67,0.00),v40,z0,tPen\WObj:=wPaper;
    MoveL Offs(pOrigin,116.93,133.35,0.00),v40,z0,tPen\WObj:=wPaper;
    MoveL Offs(pOrigin,116.18,133.46,0.00),v40,fine,tPen\WObj:=wPaper;
    MoveL Offs(pOrigin,116.18,133.46,6.00),v60,z5,tPen\WObj:=wPaper;
    MoveL Offs(pOrigin,123.62,134.41,6.00),vTravel,z5,tPen\WObj:=wPaper;
    MoveL Offs(pOrigin,123.62,134.41,0.00),v60,z0,tPen\WObj:=wPaper;
    MoveL Offs(pOrigin,124.11,134.31,0.00),v40,z0,tPen\WObj:=wPaper;
    MoveL Offs(pOrigin,124.79,132.82,0.00),v40,z0,tPen\WObj:=wPaper;
    MoveL Offs(pOrigin,124.79,132.82,0.00),v40,z0,tPen\WObj:=wPaper;
    MoveL Offs(pOrigin,124.29,132.93,0.00),v40,z0,tPen\WObj:=wPaper;
    MoveL Offs(pOrigin,124.04,133.67,0.00),v40,fine,tPen\WObj:=wPaper;
    MoveL Offs(pOrigin,124.04,133.67,6.00),v60,z5,tPen\WObj:=wPaper;
    MoveL Offs(pOrigin,122.77,137.39,6.00),vTravel,z5,tPen\WObj:=wPaper;
    MoveL Offs(pOrigin,122.77,137.39,0.00),v60,z0,tPen\WObj:=wPaper;
    MoveL Offs(pOrigin,121.67,138.66,0.00),v40,z0,tPen\WObj:=wPaper;
    MoveL Offs(pOrigin,121.18,140.79,0.00),v40,fine,tPen\WObj:=wPaper;
    MoveL Offs(pOrigin,121.18,140.79,6.00),v60,z5,tPen\WObj:=wPaper;
    MoveL Offs(pOrigin,124.15,140.04,6.00),vTravel,z5,tPen\WObj:=wPaper;
    MoveL Offs(pOrigin,124.15,140.04,0.00),v60,z0,tPen\WObj:=wPaper;
    MoveL Offs(pOrigin,123.51,138.77,0.00),v40,fine,tPen\WObj:=wPaper;
    MoveL Offs(pOrigin,123.51,138.77,6.00),v60,z5,tPen\WObj:=wPaper;
    MoveL Offs(pOrigin,131.69,135.05,6.00),vTravel,z5,tPen\WObj:=wPaper;
    MoveL Offs(pOrigin,131.69,135.05,0.00),v60,z0,tPen\WObj:=wPaper;
    MoveL Offs(pOrigin,132.97,135.90,0.00),v40,fine,tPen\WObj:=wPaper;
    MoveL Offs(pOrigin,132.97,135.90,6.00),v60,z5,tPen\WObj:=wPaper;
    MoveL Offs(pOrigin,141.15,141.32,6.00),vTravel,z5,tPen\WObj:=wPaper;
    MoveL Offs(pOrigin,141.15,141.32,0.00),v60,z0,tPen\WObj:=wPaper;
    MoveL Offs(pOrigin,141.68,139.51,0.00),v40,z0,tPen\WObj:=wPaper;
    MoveL Offs(pOrigin,144.55,138.66,0.00),v40,fine,tPen\WObj:=wPaper;
    MoveL Offs(pOrigin,144.55,138.66,6.00),v60,z5,tPen\WObj:=wPaper;
    MoveL Offs(pOrigin,143.59,142.81,6.00),vTravel,z5,tPen\WObj:=wPaper;
    MoveL Offs(pOrigin,143.59,142.81,0.00),v60,z0,tPen\WObj:=wPaper;
    MoveL Offs(pOrigin,143.91,142.38,0.00),v40,z0,tPen\WObj:=wPaper;
    MoveL Offs(pOrigin,145.40,142.17,0.00),v40,z0,tPen\WObj:=wPaper;
    MoveL Offs(pOrigin,147.95,143.34,0.00),v40,z0,tPen\WObj:=wPaper;
    MoveL Offs(pOrigin,147.95,143.34,0.00),v40,z0,tPen\WObj:=wPaper;
    MoveL Offs(pOrigin,148.59,144.61,0.00),v40,z0,tPen\WObj:=wPaper;
    MoveL Offs(pOrigin,148.59,144.61,0.00),v40,z0,tPen\WObj:=wPaper;
    MoveL Offs(pOrigin,148.80,146.63,0.00),v40,z0,tPen\WObj:=wPaper;
    MoveL Offs(pOrigin,148.38,147.06,0.00),v40,z0,tPen\WObj:=wPaper;
    MoveL Offs(pOrigin,148.38,147.06,0.00),v40,z0,tPen\WObj:=wPaper;
    MoveL Offs(pOrigin,148.48,148.33,0.00),v40,fine,tPen\WObj:=wPaper;
    MoveL Offs(pOrigin,148.48,148.33,6.00),v60,z5,tPen\WObj:=wPaper;
    MoveL Offs(pOrigin,148.16,149.50,6.00),vTravel,z5,tPen\WObj:=wPaper;
    MoveL Offs(pOrigin,148.16,149.50,0.00),v60,z0,tPen\WObj:=wPaper;
    MoveL Offs(pOrigin,148.27,151.20,0.00),v40,fine,tPen\WObj:=wPaper;
  ENDPROC

  PROC DrawPart21()
    MoveL Offs(pOrigin,148.27,151.20,6.00),v60,z5,tPen\WObj:=wPaper;
    MoveL Offs(pOrigin,146.89,152.69,6.00),vTravel,z5,tPen\WObj:=wPaper;
    MoveL Offs(pOrigin,146.89,152.69,0.00),v60,z0,tPen\WObj:=wPaper;
    MoveL Offs(pOrigin,145.93,152.37,0.00),v40,z0,tPen\WObj:=wPaper;
    MoveL Offs(pOrigin,145.93,152.37,0.00),v40,z0,tPen\WObj:=wPaper;
    MoveL Offs(pOrigin,145.61,152.05,0.00),v40,z0,tPen\WObj:=wPaper;
    MoveL Offs(pOrigin,144.34,152.19,0.00),v40,z0,tPen\WObj:=wPaper;
    MoveL Offs(pOrigin,142.74,153.64,0.00),v40,z0,tPen\WObj:=wPaper;
    MoveL Offs(pOrigin,142.53,153.75,0.00),v40,z0,tPen\WObj:=wPaper;
    MoveL Offs(pOrigin,141.36,154.64,0.00),v40,z0,tPen\WObj:=wPaper;
    MoveL Offs(pOrigin,139.24,155.24,0.00),v40,z0,tPen\WObj:=wPaper;
    MoveL Offs(pOrigin,139.24,155.24,0.00),v40,z0,tPen\WObj:=wPaper;
    MoveL Offs(pOrigin,139.45,154.81,0.00),v40,z0,tPen\WObj:=wPaper;
    MoveL Offs(pOrigin,142.96,152.48,0.00),v40,z0,tPen\WObj:=wPaper;
    MoveL Offs(pOrigin,143.17,152.37,0.00),v40,z0,tPen\WObj:=wPaper;
    MoveL Offs(pOrigin,144.66,151.16,0.00),v40,z0,tPen\WObj:=wPaper;
    MoveL Offs(pOrigin,146.25,150.46,0.00),v40,fine,tPen\WObj:=wPaper;
    MoveL Offs(pOrigin,146.25,150.46,6.00),v60,z5,tPen\WObj:=wPaper;
    MoveL Offs(pOrigin,145.93,152.37,6.00),vTravel,z5,tPen\WObj:=wPaper;
    MoveL Offs(pOrigin,145.93,152.37,0.00),v60,z0,tPen\WObj:=wPaper;
    MoveL Offs(pOrigin,145.19,152.90,0.00),v40,z0,tPen\WObj:=wPaper;
    MoveL Offs(pOrigin,144.98,153.01,0.00),v40,z0,tPen\WObj:=wPaper;
    MoveL Offs(pOrigin,144.44,153.75,0.00),v40,z0,tPen\WObj:=wPaper;
    MoveL Offs(pOrigin,144.44,153.75,0.00),v40,z0,tPen\WObj:=wPaper;
    MoveL Offs(pOrigin,143.81,153.86,0.00),v40,z0,tPen\WObj:=wPaper;
    MoveL Offs(pOrigin,143.49,154.28,0.00),v40,z0,tPen\WObj:=wPaper;
    MoveL Offs(pOrigin,144.44,154.07,0.00),v40,z0,tPen\WObj:=wPaper;
    MoveL Offs(pOrigin,143.91,155.34,0.00),v40,z0,tPen\WObj:=wPaper;
    MoveL Offs(pOrigin,143.91,155.34,0.00),v40,z0,tPen\WObj:=wPaper;
    MoveL Offs(pOrigin,143.56,156.90,0.00),v40,z0,tPen\WObj:=wPaper;
    MoveL Offs(pOrigin,142.85,157.47,0.00),v40,z0,tPen\WObj:=wPaper;
    MoveL Offs(pOrigin,143.27,158.11,0.00),v40,z0,tPen\WObj:=wPaper;
    MoveL Offs(pOrigin,142.21,158.64,0.00),v40,z0,tPen\WObj:=wPaper;
    MoveL Offs(pOrigin,141.36,158.64,0.00),v40,z0,tPen\WObj:=wPaper;
    MoveL Offs(pOrigin,138.71,157.89,0.00),v40,z0,tPen\WObj:=wPaper;
    MoveL Offs(pOrigin,137.96,158.00,0.00),v40,fine,tPen\WObj:=wPaper;
    MoveL Offs(pOrigin,137.96,158.00,6.00),v60,z5,tPen\WObj:=wPaper;
    MoveL Offs(pOrigin,137.01,156.51,6.00),vTravel,z5,tPen\WObj:=wPaper;
    MoveL Offs(pOrigin,137.01,156.51,0.00),v60,z0,tPen\WObj:=wPaper;
    MoveL Offs(pOrigin,138.39,156.62,0.00),v40,z0,tPen\WObj:=wPaper;
    MoveL Offs(pOrigin,138.92,157.04,0.00),v40,z0,tPen\WObj:=wPaper;
    MoveL Offs(pOrigin,140.94,157.47,0.00),v40,z0,tPen\WObj:=wPaper;
    MoveL Offs(pOrigin,141.68,156.62,0.00),v40,z0,tPen\WObj:=wPaper;
    MoveL Offs(pOrigin,139.24,156.41,0.00),v40,z0,tPen\WObj:=wPaper;
    MoveL Offs(pOrigin,139.24,156.41,0.00),v40,z0,tPen\WObj:=wPaper;
    MoveL Offs(pOrigin,142.11,155.13,0.00),v40,fine,tPen\WObj:=wPaper;
    MoveL Offs(pOrigin,142.11,155.13,6.00),v60,z5,tPen\WObj:=wPaper;
    MoveL Offs(pOrigin,140.19,153.32,6.00),vTravel,z5,tPen\WObj:=wPaper;
    MoveL Offs(pOrigin,140.19,153.32,0.00),v60,z0,tPen\WObj:=wPaper;
    MoveL Offs(pOrigin,140.83,153.11,0.00),v40,z0,tPen\WObj:=wPaper;
    MoveL Offs(pOrigin,143.81,150.24,0.00),v40,z0,tPen\WObj:=wPaper;
    MoveL Offs(pOrigin,143.81,149.61,0.00),v40,z0,tPen\WObj:=wPaper;
    MoveL Offs(pOrigin,142.85,149.93,0.00),v40,z0,tPen\WObj:=wPaper;
    MoveL Offs(pOrigin,139.88,152.37,0.00),v40,z0,tPen\WObj:=wPaper;
    MoveL Offs(pOrigin,139.66,152.26,0.00),v40,z0,tPen\WObj:=wPaper;
    MoveL Offs(pOrigin,139.45,151.94,0.00),v40,z0,tPen\WObj:=wPaper;
    MoveL Offs(pOrigin,139.98,151.20,0.00),v40,z0,tPen\WObj:=wPaper;
    MoveL Offs(pOrigin,142.32,149.07,0.00),v40,z0,tPen\WObj:=wPaper;
    MoveL Offs(pOrigin,144.98,147.69,0.00),v40,fine,tPen\WObj:=wPaper;
    MoveL Offs(pOrigin,144.98,147.69,6.00),v60,z5,tPen\WObj:=wPaper;
    MoveL Offs(pOrigin,143.27,147.59,6.00),vTravel,z5,tPen\WObj:=wPaper;
    MoveL Offs(pOrigin,143.27,147.59,0.00),v60,z0,tPen\WObj:=wPaper;
    MoveL Offs(pOrigin,142.32,148.12,0.00),v40,z0,tPen\WObj:=wPaper;
    MoveL Offs(pOrigin,142.11,148.23,0.00),v40,z0,tPen\WObj:=wPaper;
    MoveL Offs(pOrigin,140.51,149.50,0.00),v40,z0,tPen\WObj:=wPaper;
    MoveL Offs(pOrigin,140.41,149.50,0.00),v40,z0,tPen\WObj:=wPaper;
    MoveL Offs(pOrigin,140.62,150.46,0.00),v40,z0,tPen\WObj:=wPaper;
    MoveL Offs(pOrigin,140.41,149.50,0.00),v40,z0,tPen\WObj:=wPaper;
    MoveL Offs(pOrigin,140.83,147.91,0.00),v40,z0,tPen\WObj:=wPaper;
    MoveL Offs(pOrigin,140.62,147.69,0.00),v40,z0,tPen\WObj:=wPaper;
    MoveL Offs(pOrigin,139.34,149.18,0.00),v40,z0,tPen\WObj:=wPaper;
    MoveL Offs(pOrigin,139.45,150.14,0.00),v40,z0,tPen\WObj:=wPaper;
    MoveL Offs(pOrigin,139.63,150.46,0.00),v40,z0,tPen\WObj:=wPaper;
    MoveL Offs(pOrigin,139.13,150.99,0.00),v40,fine,tPen\WObj:=wPaper;
    MoveL Offs(pOrigin,139.13,150.99,6.00),v60,z5,tPen\WObj:=wPaper;
    MoveL Offs(pOrigin,138.71,152.26,6.00),vTravel,z5,tPen\WObj:=wPaper;
    MoveL Offs(pOrigin,138.71,152.26,0.00),v60,z0,tPen\WObj:=wPaper;
    MoveL Offs(pOrigin,137.86,152.90,0.00),v40,z0,tPen\WObj:=wPaper;
    MoveL Offs(pOrigin,138.07,153.64,0.00),v40,z0,tPen\WObj:=wPaper;
    MoveL Offs(pOrigin,136.37,154.28,0.00),v40,fine,tPen\WObj:=wPaper;
    MoveL Offs(pOrigin,136.37,154.28,6.00),v60,z5,tPen\WObj:=wPaper;
    MoveL Offs(pOrigin,135.52,155.13,6.00),vTravel,z5,tPen\WObj:=wPaper;
    MoveL Offs(pOrigin,135.52,155.13,0.00),v60,z0,tPen\WObj:=wPaper;
    MoveL Offs(pOrigin,137.75,154.42,0.00),v40,z0,tPen\WObj:=wPaper;
    MoveL Offs(pOrigin,138.07,154.71,0.00),v40,z0,tPen\WObj:=wPaper;
    MoveL Offs(pOrigin,138.39,155.24,0.00),v40,z0,tPen\WObj:=wPaper;
    MoveL Offs(pOrigin,138.07,153.86,0.00),v40,z0,tPen\WObj:=wPaper;
    MoveL Offs(pOrigin,139.06,152.69,0.00),v40,z0,tPen\WObj:=wPaper;
    MoveL Offs(pOrigin,138.92,152.37,0.00),v40,fine,tPen\WObj:=wPaper;
    MoveL Offs(pOrigin,138.92,152.37,6.00),v60,z5,tPen\WObj:=wPaper;
    MoveL Offs(pOrigin,140.19,153.32,6.00),vTravel,z5,tPen\WObj:=wPaper;
    MoveL Offs(pOrigin,140.19,153.32,0.00),v60,z0,tPen\WObj:=wPaper;
    MoveL Offs(pOrigin,140.83,152.26,0.00),v40,fine,tPen\WObj:=wPaper;
    MoveL Offs(pOrigin,140.83,152.26,6.00),v60,z5,tPen\WObj:=wPaper;
    MoveL Offs(pOrigin,142.00,150.56,6.00),vTravel,z5,tPen\WObj:=wPaper;
    MoveL Offs(pOrigin,142.00,150.56,0.00),v60,z0,tPen\WObj:=wPaper;
    MoveL Offs(pOrigin,141.26,151.31,0.00),v40,z0,tPen\WObj:=wPaper;
    MoveL Offs(pOrigin,142.00,150.56,0.00),v40,z0,tPen\WObj:=wPaper;
    MoveL Offs(pOrigin,141.68,149.61,0.00),v40,z0,tPen\WObj:=wPaper;
    MoveL Offs(pOrigin,141.36,149.93,0.00),v40,z0,tPen\WObj:=wPaper;
    MoveL Offs(pOrigin,141.68,149.61,0.00),v40,z0,tPen\WObj:=wPaper;
    MoveL Offs(pOrigin,142.85,149.82,0.00),v40,z0,tPen\WObj:=wPaper;
    MoveL Offs(pOrigin,142.32,150.35,0.00),v40,z0,tPen\WObj:=wPaper;
    MoveL Offs(pOrigin,142.85,149.82,0.00),v40,fine,tPen\WObj:=wPaper;
    MoveL Offs(pOrigin,142.85,149.82,6.00),v60,z5,tPen\WObj:=wPaper;
    MoveL Offs(pOrigin,141.47,146.95,6.00),vTravel,z5,tPen\WObj:=wPaper;
    MoveL Offs(pOrigin,141.47,146.95,0.00),v60,z0,tPen\WObj:=wPaper;
    MoveL Offs(pOrigin,141.47,146.42,0.00),v40,z0,tPen\WObj:=wPaper;
    MoveL Offs(pOrigin,142.00,146.21,0.00),v40,fine,tPen\WObj:=wPaper;
    MoveL Offs(pOrigin,142.00,146.21,6.00),v60,z5,tPen\WObj:=wPaper;
    MoveL Offs(pOrigin,141.47,145.04,6.00),vTravel,z5,tPen\WObj:=wPaper;
    MoveL Offs(pOrigin,141.47,145.04,0.00),v60,z0,tPen\WObj:=wPaper;
    MoveL Offs(pOrigin,142.64,144.51,0.00),v40,z0,tPen\WObj:=wPaper;
    MoveL Offs(pOrigin,142.85,144.40,0.00),v40,z0,tPen\WObj:=wPaper;
    MoveL Offs(pOrigin,145.29,143.34,0.00),v40,fine,tPen\WObj:=wPaper;
    MoveL Offs(pOrigin,145.29,143.34,6.00),v60,z5,tPen\WObj:=wPaper;
    MoveL Offs(pOrigin,143.59,142.81,6.00),vTravel,z5,tPen\WObj:=wPaper;
    MoveL Offs(pOrigin,143.59,142.81,0.00),v60,z0,tPen\WObj:=wPaper;
    MoveL Offs(pOrigin,145.08,143.02,0.00),v40,z0,tPen\WObj:=wPaper;
    MoveL Offs(pOrigin,148.59,144.61,0.00),v40,fine,tPen\WObj:=wPaper;
  ENDPROC

  PROC DrawPart22()
    MoveL Offs(pOrigin,148.59,144.61,6.00),v60,z5,tPen\WObj:=wPaper;
    MoveL Offs(pOrigin,147.95,146.95,6.00),vTravel,z5,tPen\WObj:=wPaper;
    MoveL Offs(pOrigin,147.95,146.95,0.00),v60,z0,tPen\WObj:=wPaper;
    MoveL Offs(pOrigin,146.46,146.31,0.00),v40,fine,tPen\WObj:=wPaper;
    MoveL Offs(pOrigin,146.46,146.31,6.00),v60,z5,tPen\WObj:=wPaper;
    MoveL Offs(pOrigin,148.38,147.06,6.00),vTravel,z5,tPen\WObj:=wPaper;
    MoveL Offs(pOrigin,148.38,147.06,0.00),v60,z0,tPen\WObj:=wPaper;
    MoveL Offs(pOrigin,147.99,146.84,0.00),v40,z0,tPen\WObj:=wPaper;
    MoveL Offs(pOrigin,147.52,145.57,0.00),v40,z0,tPen\WObj:=wPaper;
    MoveL Offs(pOrigin,146.25,144.82,0.00),v40,z0,tPen\WObj:=wPaper;
    MoveL Offs(pOrigin,144.66,144.72,0.00),v40,z0,tPen\WObj:=wPaper;
    MoveL Offs(pOrigin,143.70,145.07,0.00),v40,z0,tPen\WObj:=wPaper;
    MoveL Offs(pOrigin,143.49,145.46,0.00),v40,fine,tPen\WObj:=wPaper;
    MoveL Offs(pOrigin,143.49,145.46,6.00),v60,z5,tPen\WObj:=wPaper;
    MoveL Offs(pOrigin,141.36,145.04,6.00),vTravel,z5,tPen\WObj:=wPaper;
    MoveL Offs(pOrigin,141.36,145.04,0.00),v60,z0,tPen\WObj:=wPaper;
    MoveL Offs(pOrigin,140.62,145.36,0.00),v40,z0,tPen\WObj:=wPaper;
    MoveL Offs(pOrigin,139.34,147.06,0.00),v40,z0,tPen\WObj:=wPaper;
    MoveL Offs(pOrigin,139.77,147.80,0.00),v40,z0,tPen\WObj:=wPaper;
    MoveL Offs(pOrigin,140.62,146.74,0.00),v40,fine,tPen\WObj:=wPaper;
    MoveL Offs(pOrigin,140.62,146.74,6.00),v60,z5,tPen\WObj:=wPaper;
    MoveL Offs(pOrigin,139.56,143.87,6.00),vTravel,z5,tPen\WObj:=wPaper;
    MoveL Offs(pOrigin,139.56,143.87,0.00),v60,z0,tPen\WObj:=wPaper;
    MoveL Offs(pOrigin,140.26,142.59,0.00),v40,z0,tPen\WObj:=wPaper;
    MoveL Offs(pOrigin,140.73,142.38,0.00),v40,fine,tPen\WObj:=wPaper;
    MoveL Offs(pOrigin,140.73,142.38,6.00),v60,z5,tPen\WObj:=wPaper;
    MoveL Offs(pOrigin,143.91,133.46,6.00),vTravel,z5,tPen\WObj:=wPaper;
    MoveL Offs(pOrigin,143.91,133.46,0.00),v60,z0,tPen\WObj:=wPaper;
    MoveL Offs(pOrigin,143.91,131.97,0.00),v40,fine,tPen\WObj:=wPaper;
    MoveL Offs(pOrigin,143.91,131.97,6.00),v60,z5,tPen\WObj:=wPaper;
    MoveL Offs(pOrigin,149.12,131.76,6.00),vTravel,z5,tPen\WObj:=wPaper;
    MoveL Offs(pOrigin,149.12,131.76,0.00),v60,z0,tPen\WObj:=wPaper;
    MoveL Offs(pOrigin,148.27,135.26,0.00),v40,fine,tPen\WObj:=wPaper;
    MoveL Offs(pOrigin,148.27,135.26,6.00),v60,z5,tPen\WObj:=wPaper;
    MoveL Offs(pOrigin,149.33,125.38,6.00),vTravel,z5,tPen\WObj:=wPaper;
    MoveL Offs(pOrigin,149.33,125.38,0.00),v60,z0,tPen\WObj:=wPaper;
    MoveL Offs(pOrigin,148.62,122.72,0.00),v40,z0,tPen\WObj:=wPaper;
    MoveL Offs(pOrigin,147.31,121.66,0.00),v40,z0,tPen\WObj:=wPaper;
    MoveL Offs(pOrigin,145.72,121.77,0.00),v40,fine,tPen\WObj:=wPaper;
    MoveL Offs(pOrigin,145.72,121.77,6.00),v60,z5,tPen\WObj:=wPaper;
    MoveL Offs(pOrigin,148.59,122.51,6.00),vTravel,z5,tPen\WObj:=wPaper;
    MoveL Offs(pOrigin,148.59,122.51,0.00),v60,z0,tPen\WObj:=wPaper;
    MoveL Offs(pOrigin,161.55,122.19,0.00),v40,z0,tPen\WObj:=wPaper;
    MoveL Offs(pOrigin,176.00,120.81,0.00),v40,z0,tPen\WObj:=wPaper;
    MoveL Offs(pOrigin,181.63,119.57,0.00),v40,z0,tPen\WObj:=wPaper;
    MoveL Offs(pOrigin,184.18,118.26,0.00),v40,z0,tPen\WObj:=wPaper;
    MoveL Offs(pOrigin,186.02,116.24,0.00),v40,z0,tPen\WObj:=wPaper;
    MoveL Offs(pOrigin,187.26,113.16,0.00),v40,z0,tPen\WObj:=wPaper;
    MoveL Offs(pOrigin,187.79,109.55,0.00),v40,z0,tPen\WObj:=wPaper;
    MoveL Offs(pOrigin,188.32,109.02,0.00),v40,fine,tPen\WObj:=wPaper;
    MoveL Offs(pOrigin,188.32,109.02,6.00),v60,z5,tPen\WObj:=wPaper;
    MoveL Offs(pOrigin,186.52,97.44,6.00),vTravel,z5,tPen\WObj:=wPaper;
    MoveL Offs(pOrigin,186.52,97.44,0.00),v60,z0,tPen\WObj:=wPaper;
    MoveL Offs(pOrigin,187.76,96.59,0.00),v40,z0,tPen\WObj:=wPaper;
    MoveL Offs(pOrigin,188.22,95.74,0.00),v40,z0,tPen\WObj:=wPaper;
    MoveL Offs(pOrigin,186.16,91.91,0.00),v40,z0,tPen\WObj:=wPaper;
    MoveL Offs(pOrigin,185.14,89.04,0.00),v40,fine,tPen\WObj:=wPaper;
    MoveL Offs(pOrigin,185.14,89.04,6.00),v60,z5,tPen\WObj:=wPaper;
    MoveL Offs(pOrigin,185.35,97.44,6.00),vTravel,z5,tPen\WObj:=wPaper;
    MoveL Offs(pOrigin,185.35,97.44,0.00),v60,z0,tPen\WObj:=wPaper;
    MoveL Offs(pOrigin,183.33,98.29,0.00),v40,z0,tPen\WObj:=wPaper;
    MoveL Offs(pOrigin,169.20,102.29,0.00),v40,z0,tPen\WObj:=wPaper;
    MoveL Offs(pOrigin,155.60,107.64,0.00),v40,z0,tPen\WObj:=wPaper;
    MoveL Offs(pOrigin,151.67,108.70,0.00),v40,z0,tPen\WObj:=wPaper;
    MoveL Offs(pOrigin,151.07,108.59,0.00),v40,z0,tPen\WObj:=wPaper;
    MoveL Offs(pOrigin,151.24,107.96,0.00),v40,z0,tPen\WObj:=wPaper;
    MoveL Offs(pOrigin,154.01,104.70,0.00),v40,z0,tPen\WObj:=wPaper;
    MoveL Offs(pOrigin,155.39,104.77,0.00),v40,z0,tPen\WObj:=wPaper;
    MoveL Offs(pOrigin,158.15,104.13,0.00),v40,z0,tPen\WObj:=wPaper;
    MoveL Offs(pOrigin,167.18,101.05,0.00),v40,fine,tPen\WObj:=wPaper;
    MoveL Offs(pOrigin,167.18,101.05,6.00),v60,z5,tPen\WObj:=wPaper;
    MoveL Offs(pOrigin,146.99,55.47,6.00),vTravel,z5,tPen\WObj:=wPaper;
    MoveL Offs(pOrigin,146.99,55.47,0.00),v60,z0,tPen\WObj:=wPaper;
    MoveL Offs(pOrigin,145.93,51.54,0.00),v40,z0,tPen\WObj:=wPaper;
    MoveL Offs(pOrigin,145.93,51.54,0.00),v40,z0,tPen\WObj:=wPaper;
    MoveL Offs(pOrigin,143.81,43.25,0.00),v40,z0,tPen\WObj:=wPaper;
    MoveL Offs(pOrigin,142.74,36.38,0.00),v40,z0,tPen\WObj:=wPaper;
    MoveL Offs(pOrigin,140.94,36.45,0.00),v40,z0,tPen\WObj:=wPaper;
    MoveL Offs(pOrigin,137.64,35.49,0.00),v40,z0,tPen\WObj:=wPaper;
    MoveL Offs(pOrigin,136.37,42.72,0.00),v40,fine,tPen\WObj:=wPaper;
    MoveL Offs(pOrigin,136.37,42.72,6.00),v60,z5,tPen\WObj:=wPaper;
    MoveL Offs(pOrigin,137.64,35.39,6.00),vTravel,z5,tPen\WObj:=wPaper;
    MoveL Offs(pOrigin,137.64,35.39,0.00),v60,z0,tPen\WObj:=wPaper;
    MoveL Offs(pOrigin,135.09,33.90,0.00),v40,z0,tPen\WObj:=wPaper;
    MoveL Offs(pOrigin,135.09,33.90,0.00),v40,z0,tPen\WObj:=wPaper;
    MoveL Offs(pOrigin,132.12,32.77,0.00),v40,z0,tPen\WObj:=wPaper;
    MoveL Offs(pOrigin,128.93,30.82,0.00),v40,z0,tPen\WObj:=wPaper;
    MoveL Offs(pOrigin,124.47,26.46,0.00),v40,z0,tPen\WObj:=wPaper;
    MoveL Offs(pOrigin,121.07,22.32,0.00),v40,z0,tPen\WObj:=wPaper;
    MoveL Offs(pOrigin,121.07,22.32,0.00),v40,z0,tPen\WObj:=wPaper;
    MoveL Offs(pOrigin,120.96,21.15,0.00),v40,z0,tPen\WObj:=wPaper;
    MoveL Offs(pOrigin,121.35,20.30,0.00),v40,z0,tPen\WObj:=wPaper;
    MoveL Offs(pOrigin,122.34,19.88,0.00),v40,z0,tPen\WObj:=wPaper;
    MoveL Offs(pOrigin,122.34,19.88,0.00),v40,z0,tPen\WObj:=wPaper;
    MoveL Offs(pOrigin,123.41,21.58,0.00),v40,z0,tPen\WObj:=wPaper;
    MoveL Offs(pOrigin,127.12,24.55,0.00),v40,z0,tPen\WObj:=wPaper;
    MoveL Offs(pOrigin,132.23,28.09,0.00),v40,z0,tPen\WObj:=wPaper;
    MoveL Offs(pOrigin,135.31,29.65,0.00),v40,z0,tPen\WObj:=wPaper;
    MoveL Offs(pOrigin,135.31,29.65,0.00),v40,z0,tPen\WObj:=wPaper;
    MoveL Offs(pOrigin,134.81,31.14,0.00),v40,z0,tPen\WObj:=wPaper;
    MoveL Offs(pOrigin,133.18,33.05,0.00),v40,z0,tPen\WObj:=wPaper;
    MoveL Offs(pOrigin,133.71,33.37,0.00),v40,z0,tPen\WObj:=wPaper;
    MoveL Offs(pOrigin,135.34,31.14,0.00),v40,z0,tPen\WObj:=wPaper;
    MoveL Offs(pOrigin,135.62,29.97,0.00),v40,z0,tPen\WObj:=wPaper;
    MoveL Offs(pOrigin,135.31,29.65,0.00),v40,z0,tPen\WObj:=wPaper;
    MoveL Offs(pOrigin,135.62,29.76,0.00),v40,z0,tPen\WObj:=wPaper;
    MoveL Offs(pOrigin,136.58,30.08,0.00),v40,z0,tPen\WObj:=wPaper;
    MoveL Offs(pOrigin,136.58,30.08,0.00),v40,z0,tPen\WObj:=wPaper;
    MoveL Offs(pOrigin,135.55,32.41,0.00),v40,z0,tPen\WObj:=wPaper;
    MoveL Offs(pOrigin,134.77,33.16,0.00),v40,z0,tPen\WObj:=wPaper;
    MoveL Offs(pOrigin,135.09,33.90,0.00),v40,z0,tPen\WObj:=wPaper;
    MoveL Offs(pOrigin,136.19,32.41,0.00),v40,z0,tPen\WObj:=wPaper;
    MoveL Offs(pOrigin,137.01,30.18,0.00),v40,z0,tPen\WObj:=wPaper;
    MoveL Offs(pOrigin,137.01,30.18,0.00),v40,z0,tPen\WObj:=wPaper;
    MoveL Offs(pOrigin,139.45,31.00,0.00),v40,z0,tPen\WObj:=wPaper;
    MoveL Offs(pOrigin,140.94,32.09,0.00),v40,fine,tPen\WObj:=wPaper;
    MoveL Offs(pOrigin,140.94,32.09,6.00),v60,z5,tPen\WObj:=wPaper;
    MoveL Offs(pOrigin,142.85,36.34,6.00),vTravel,z5,tPen\WObj:=wPaper;
    MoveL Offs(pOrigin,142.85,36.34,0.00),v60,z0,tPen\WObj:=wPaper;
    MoveL Offs(pOrigin,146.46,34.29,0.00),v40,z0,tPen\WObj:=wPaper;
  ENDPROC

